// TIA Portal V16 export
// export: Created 2024-05-11T02:56:22.8632211Z, ExportSetting WithDefaults, DisplayName Totally Integrated Automation Portal, DisplayVersion V16, DisplayName TIA Portal Version Control Interface, DisplayVersion V16, DisplayName TIA Portal Openness, DisplayVersion V16, DisplayName STEP 7 Professional, DisplayVersion V16, DisplayName STEP 7 Safety, DisplayVersion V16, DisplayName WinCC Professional, DisplayVersion V16
FUNCTION_BLOCK "K06_动作"   // FB6, LAD
{ S7_Optimized_Access := 'TRUE' }
VERSION : 0.1
// stored: AutoNumber false, IsIECCheckEnabled false, IsRetainMemResEnabled false, MemoryReserve 100, SetENOAutomatically false, UDAEnableTagReadback false
   VAR
      INV_Time1 : IEC_TIMER;
      INV_Time2 : IEC_TIMER;
      F100_Val_Instance1 { S7_SetPoint := 'True'} : "F100_Val";   // EN阻挡
      F100_Val_Instance2 { S7_SetPoint := 'True'} : "F100_Val";   // EN提升机
      F100_Val_Instance3 { S7_SetPoint := 'True'} : "F100_Val";   // EX阻挡
      F100_Val_Instance4 { S7_SetPoint := 'True'} : "F100_Val";   // EX提升机
      F100_Val_Instance5 { S7_SetPoint := 'True'} : "F100_Val";   // ST01上阻挡
      F100_Val_Instance6 { S7_SetPoint := 'True'} : "F100_Val";   // ST01下阻挡
      F100_Val_Instance7 { S7_SetPoint := 'True'} : "F100_Val";   // ST02上阻挡
      F100_Val_Instance8 { S7_SetPoint := 'True'} : "F100_Val";   // ST02下阻挡
      F100_Val_Instance9 { S7_SetPoint := 'True'} : "F100_Val";   // ST03上阻挡
      F100_Val_Instance10 { S7_SetPoint := 'True'} : "F100_Val";   // ST03下阻挡
      F100_Val_Instance11 { S7_SetPoint := 'True'} : "F100_Val";   // ST04上阻挡
      F100_Val_Instance12 { S7_SetPoint := 'True'} : "F100_Val";   // ST05上阻挡
      F100_Val_Instance13 { S7_SetPoint := 'True'} : "F100_Val";   // ST06上阻挡
      F100_Val_Instance14 { S7_SetPoint := 'True'} : "F100_Val";   // ST07上阻挡
      F100_Val_Instance15 { S7_SetPoint := 'True'} : "F100_Val";   // ST08上阻挡
      F100_Val_Instance16 { S7_SetPoint := 'True'} : "F100_Val";   // ST09上阻挡
      F100_Val_Instance17 { S7_SetPoint := 'True'} : "F100_Val";   // ST10上阻挡
      F100_Val_Instance18 { S7_SetPoint := 'True'} : "F100_Val";   // ST11上阻挡
      F100_Val_Instance19 { S7_SetPoint := 'True'} : "F100_Val";   // ST12上阻挡
      F110_Inv_Instance1 { S7_SetPoint := 'True'} : "F110_Inv";   // 入口变频器
      F110_Inv_Instance2 { S7_SetPoint := 'True'} : "F110_Inv";   // 出口变频器
      F110_Inv_Instance3 { S7_SetPoint := 'True'} : "F110_Inv";   // 上层线体变频器
      F110_Inv_Instance4 { S7_SetPoint := 'True'} : "F110_Inv";   // 下层线体变频器
   END_VAR
   VAR_TEMP
      M_Pluse : Array[1..20] of Bool;
      上线体正转 : Bool;
      上线体反转 : Bool;
      上线体高速 : Bool;
      上线体低速 : Bool;
      上线体复位 : Bool;
      下线体正转 : Bool;
      下线体反转 : Bool;
      下线体高速 : Bool;
      下线体低速 : Bool;
      下线体复位 : Bool;
   END_VAR
   VAR_TEMP   // added for the SCL form of the ladder/FBD networks
      _w1 : Bool;
      _w2 : Bool;
      _w3 : Bool;
      _w4 : Bool;
      _w5 : Bool;
      _w6 : Bool;
      _w7 : Bool;
      _w8 : Bool;
      _w9 : Bool;
      _w10 : Bool;
      _w11 : Bool;
      _w12 : Bool;
   END_VAR
BEGIN

REGION Network 1: 阀1 入口阻挡
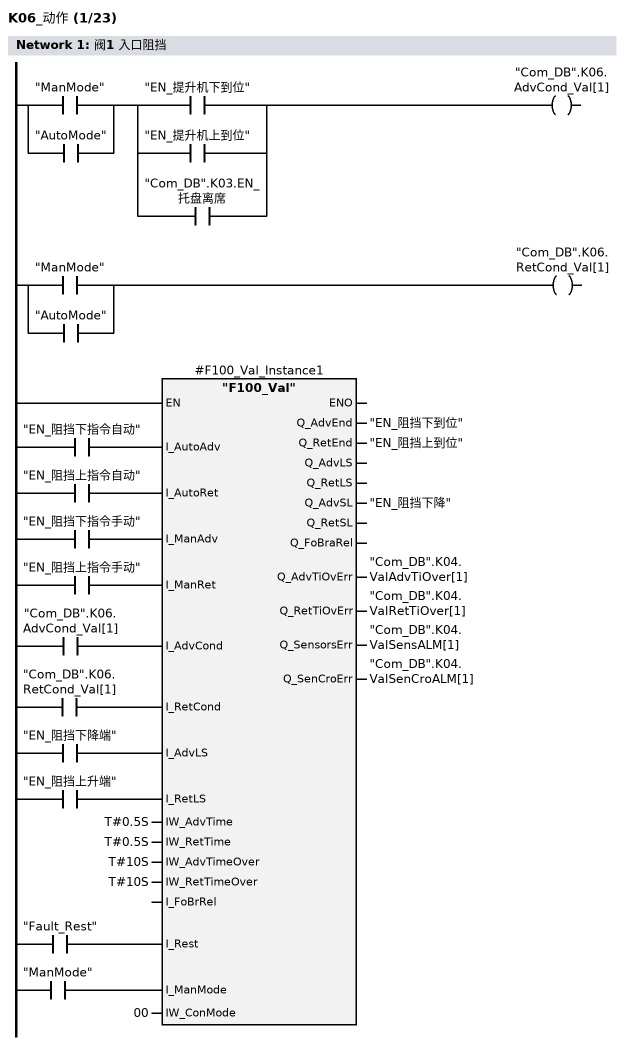
   RUNG wire#powerrail
      Contact( "ManMode" )
      wire#w1
      Contact( "EN_提升机下到位" )
      wire#w2
      Coil( "Com_DB".K06.AdvCond_Val[1] )
   END_RUNG
   RUNG wire#powerrail
      Contact( "AutoMode" )
   END_RUNG wire#w1
   RUNG wire#w1
      Contact( "EN_提升机上到位" )
   END_RUNG wire#w2
   RUNG wire#w1
      Contact( "Com_DB".K03.EN_托盘离席 )
   END_RUNG wire#w2
   RUNG wire#powerrail
      Contact( "ManMode" )
      wire#w3
      Coil( "Com_DB".K06.RetCond_Val[1] )
   END_RUNG
   RUNG wire#powerrail
      Contact( "AutoMode" )
   END_RUNG wire#w3
   RUNG wire#powerrail
      #F100_Val_Instance1(I_AutoAdv := wire#w4, I_AutoRet := wire#w5, I_ManAdv := wire#w6, I_ManRet := wire#w7, I_AdvCond := wire#w8, I_RetCond := wire#w9, I_AdvLS := wire#w10, I_RetLS := wire#w11, I_Rest := wire#w12, I_ManMode := wire#w13, IW_AdvTime := T#0.5S, IW_RetTime := T#0.5S, IW_AdvTimeOver := T#10S, IW_RetTimeOver := T#10S, I_FoBrRel :=, IW_ConMode := 00, Q_AdvEnd => "EN_阻挡下到位", Q_RetEnd => "EN_阻挡上到位", Q_AdvLS =>, Q_RetLS =>, Q_AdvSL => "EN_阻挡下降", Q_RetSL =>, Q_FoBraRel =>, Q_AdvTiOvErr => "Com_DB".K04.ValAdvTiOver[1], Q_RetTiOvErr => "Com_DB".K04.ValRetTiOver[1], Q_SensorsErr => "Com_DB".K04.ValSensALM[1], Q_SenCroErr => "Com_DB".K04.ValSenCroALM[1])
   END_RUNG
   RUNG wire#powerrail
      Contact( "EN_阻挡下指令自动" )
   END_RUNG wire#w4
   RUNG wire#powerrail
      Contact( "EN_阻挡上指令自动" )
   END_RUNG wire#w5
   RUNG wire#powerrail
      Contact( "EN_阻挡下指令手动" )
   END_RUNG wire#w6
   RUNG wire#powerrail
      Contact( "EN_阻挡上指令手动" )
   END_RUNG wire#w7
   RUNG wire#powerrail
      Contact( "Com_DB".K06.AdvCond_Val[1] )
   END_RUNG wire#w8
   RUNG wire#powerrail
      Contact( "Com_DB".K06.RetCond_Val[1] )
   END_RUNG wire#w9
   RUNG wire#powerrail
      Contact( "EN_阻挡下降端" )
   END_RUNG wire#w10
   RUNG wire#powerrail
      Contact( "EN_阻挡上升端" )
   END_RUNG wire#w11
   RUNG wire#powerrail
      Contact( "Fault_Rest" )
   END_RUNG wire#w12
   RUNG wire#powerrail
      Contact( "ManMode" )
   END_RUNG wire#w13
   // the same network as SCL:
   "Com_DB".K06.AdvCond_Val[1] := ("ManMode" OR "AutoMode") AND ("EN_提升机下到位" OR "EN_提升机上到位" OR "Com_DB".K03.EN_托盘离席);
   "Com_DB".K06.RetCond_Val[1] := "ManMode" OR "AutoMode";
   #F100_Val_Instance1(I_AutoAdv := "EN_阻挡下指令自动",   // "F100_Val"
                       I_AutoRet := "EN_阻挡上指令自动",
                       I_ManAdv := "EN_阻挡下指令手动",
                       I_ManRet := "EN_阻挡上指令手动",
                       I_AdvCond := "Com_DB".K06.AdvCond_Val[1],
                       I_RetCond := "Com_DB".K06.RetCond_Val[1],
                       I_AdvLS := "EN_阻挡下降端",
                       I_RetLS := "EN_阻挡上升端",
                       IW_AdvTime := T#0.5S,
                       IW_RetTime := T#0.5S,
                       IW_AdvTimeOver := T#10S,
                       IW_RetTimeOver := T#10S,
                       I_Rest := "Fault_Rest",
                       I_ManMode := "ManMode",
                       IW_ConMode := 00,
                       Q_AdvEnd => "EN_阻挡下到位",
                       Q_RetEnd => "EN_阻挡上到位",
                       Q_AdvSL => "EN_阻挡下降",
                       Q_AdvTiOvErr => "Com_DB".K04.ValAdvTiOver[1],
                       Q_RetTiOvErr => "Com_DB".K04.ValRetTiOver[1],
                       Q_SensorsErr => "Com_DB".K04.ValSensALM[1],
                       Q_SenCroErr => "Com_DB".K04.ValSenCroALM[1]);
END_REGION

REGION Network 2: 阀2 入口提升机
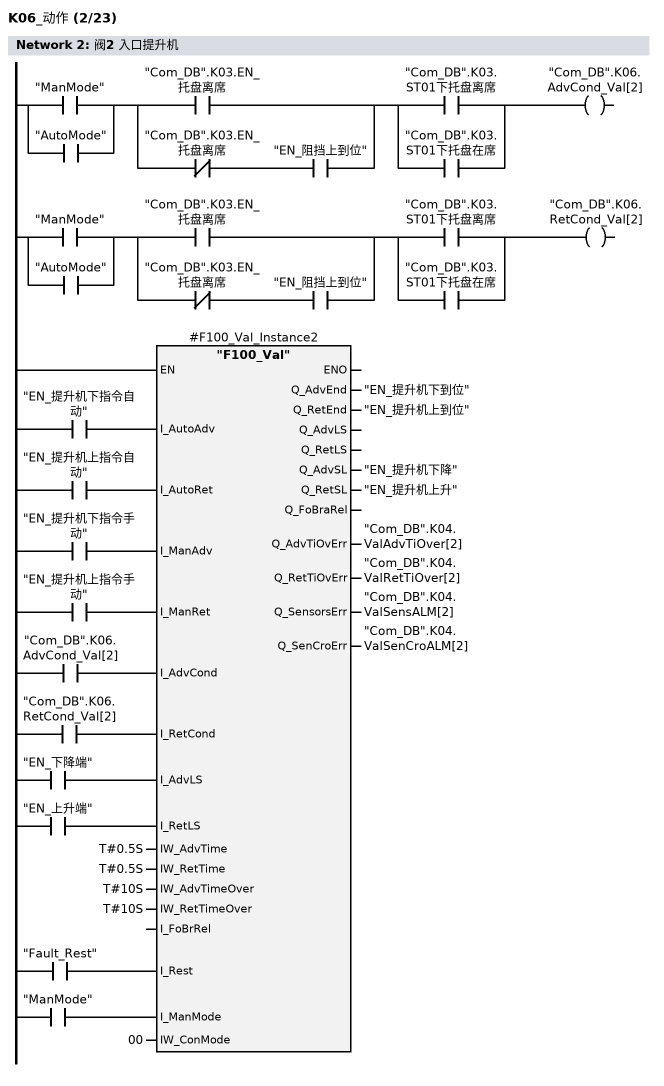
   RUNG wire#powerrail
      Contact( "ManMode" )
      wire#w1
      Contact( "Com_DB".K03.EN_托盘离席 )
      wire#w2
      Contact( "Com_DB".K03.ST01下托盘离席 )
      wire#w3
      Coil( "Com_DB".K06.AdvCond_Val[2] )
   END_RUNG
   RUNG wire#powerrail
      Contact( "AutoMode" )
   END_RUNG wire#w1
   RUNG wire#w1
      I_Contact( "Com_DB".K03.EN_托盘离席 )
      Contact( "EN_阻挡上到位" )
   END_RUNG wire#w2
   RUNG wire#w2
      Contact( "Com_DB".K03.ST01下托盘在席 )
   END_RUNG wire#w3
   RUNG wire#powerrail
      Contact( "ManMode" )
      wire#w4
      Contact( "Com_DB".K03.EN_托盘离席 )
      wire#w5
      Contact( "Com_DB".K03.ST01下托盘离席 )
      wire#w6
      Coil( "Com_DB".K06.RetCond_Val[2] )
   END_RUNG
   RUNG wire#powerrail
      Contact( "AutoMode" )
   END_RUNG wire#w4
   RUNG wire#w4
      I_Contact( "Com_DB".K03.EN_托盘离席 )
      Contact( "EN_阻挡上到位" )
   END_RUNG wire#w5
   RUNG wire#w5
      Contact( "Com_DB".K03.ST01下托盘在席 )
   END_RUNG wire#w6
   RUNG wire#powerrail
      #F100_Val_Instance2(I_AutoAdv := wire#w7, I_AutoRet := wire#w8, I_ManAdv := wire#w9, I_ManRet := wire#w10, I_AdvCond := wire#w11, I_RetCond := wire#w12, I_AdvLS := wire#w13, I_RetLS := wire#w14, I_Rest := wire#w15, I_ManMode := wire#w16, IW_AdvTime := T#0.5S, IW_RetTime := T#0.5S, IW_AdvTimeOver := T#10S, IW_RetTimeOver := T#10S, I_FoBrRel :=, IW_ConMode := 00, Q_AdvEnd => "EN_提升机下到位", Q_RetEnd => "EN_提升机上到位", Q_AdvLS =>, Q_RetLS =>, Q_AdvSL => "EN_提升机下降", Q_RetSL => "EN_提升机上升", Q_FoBraRel =>, Q_AdvTiOvErr => "Com_DB".K04.ValAdvTiOver[2], Q_RetTiOvErr => "Com_DB".K04.ValRetTiOver[2], Q_SensorsErr => "Com_DB".K04.ValSensALM[2], Q_SenCroErr => "Com_DB".K04.ValSenCroALM[2])
   END_RUNG
   RUNG wire#powerrail
      Contact( "EN_提升机下指令自动" )
   END_RUNG wire#w7
   RUNG wire#powerrail
      Contact( "EN_提升机上指令自动" )
   END_RUNG wire#w8
   RUNG wire#powerrail
      Contact( "EN_提升机下指令手动" )
   END_RUNG wire#w9
   RUNG wire#powerrail
      Contact( "EN_提升机上指令手动" )
   END_RUNG wire#w10
   RUNG wire#powerrail
      Contact( "Com_DB".K06.AdvCond_Val[2] )
   END_RUNG wire#w11
   RUNG wire#powerrail
      Contact( "Com_DB".K06.RetCond_Val[2] )
   END_RUNG wire#w12
   RUNG wire#powerrail
      Contact( "EN_下降端" )
   END_RUNG wire#w13
   RUNG wire#powerrail
      Contact( "EN_上升端" )
   END_RUNG wire#w14
   RUNG wire#powerrail
      Contact( "Fault_Rest" )
   END_RUNG wire#w15
   RUNG wire#powerrail
      Contact( "ManMode" )
   END_RUNG wire#w16
   // the same network as SCL:
   "Com_DB".K06.AdvCond_Val[2] := ("ManMode" OR "AutoMode") AND ("Com_DB".K03.EN_托盘离席 OR (NOT "Com_DB".K03.EN_托盘离席 AND "EN_阻挡上到位")) AND ("Com_DB".K03.ST01下托盘离席 OR "Com_DB".K03.ST01下托盘在席);
   "Com_DB".K06.RetCond_Val[2] := ("ManMode" OR "AutoMode") AND ("Com_DB".K03.EN_托盘离席 OR (NOT "Com_DB".K03.EN_托盘离席 AND "EN_阻挡上到位")) AND ("Com_DB".K03.ST01下托盘离席 OR "Com_DB".K03.ST01下托盘在席);
   #F100_Val_Instance2(I_AutoAdv := "EN_提升机下指令自动",   // "F100_Val"
                       I_AutoRet := "EN_提升机上指令自动",
                       I_ManAdv := "EN_提升机下指令手动",
                       I_ManRet := "EN_提升机上指令手动",
                       I_AdvCond := "Com_DB".K06.AdvCond_Val[2],
                       I_RetCond := "Com_DB".K06.RetCond_Val[2],
                       I_AdvLS := "EN_下降端",
                       I_RetLS := "EN_上升端",
                       IW_AdvTime := T#0.5S,
                       IW_RetTime := T#0.5S,
                       IW_AdvTimeOver := T#10S,
                       IW_RetTimeOver := T#10S,
                       I_Rest := "Fault_Rest",
                       I_ManMode := "ManMode",
                       IW_ConMode := 00,
                       Q_AdvEnd => "EN_提升机下到位",
                       Q_RetEnd => "EN_提升机上到位",
                       Q_AdvSL => "EN_提升机下降",
                       Q_RetSL => "EN_提升机上升",
                       Q_AdvTiOvErr => "Com_DB".K04.ValAdvTiOver[2],
                       Q_RetTiOvErr => "Com_DB".K04.ValRetTiOver[2],
                       Q_SensorsErr => "Com_DB".K04.ValSensALM[2],
                       Q_SenCroErr => "Com_DB".K04.ValSenCroALM[2]);
END_REGION

REGION Network 3: 阀3 出口阻挡
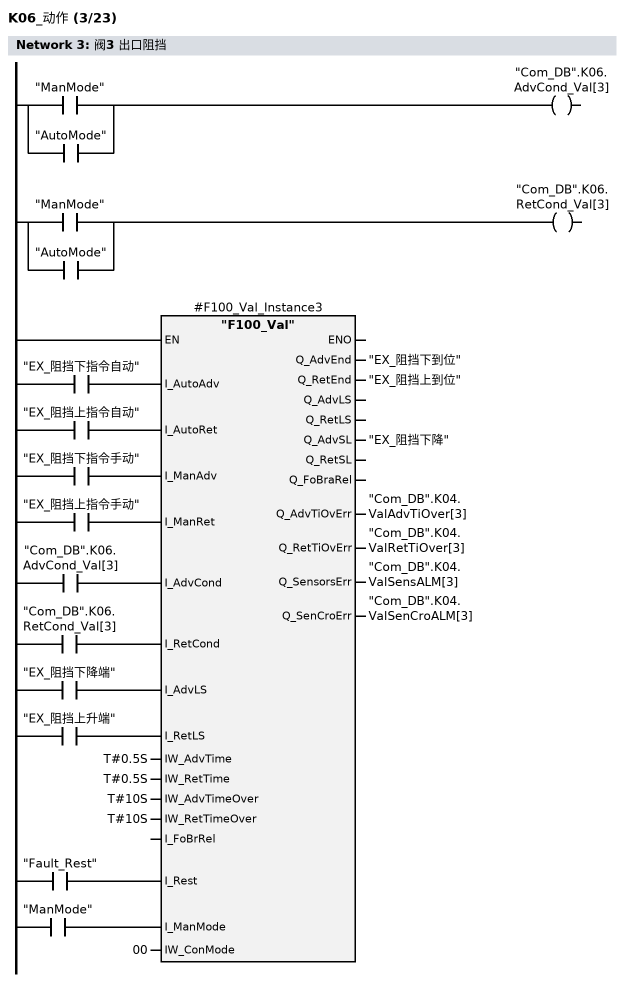
   RUNG wire#powerrail
      Contact( "ManMode" )
      wire#w1
      Coil( "Com_DB".K06.AdvCond_Val[3] )
   END_RUNG
   RUNG wire#powerrail
      Contact( "AutoMode" )
   END_RUNG wire#w1
   RUNG wire#powerrail
      Contact( "ManMode" )
      wire#w2
      Coil( "Com_DB".K06.RetCond_Val[3] )
   END_RUNG
   RUNG wire#powerrail
      Contact( "AutoMode" )
   END_RUNG wire#w2
   RUNG wire#powerrail
      #F100_Val_Instance3(I_AutoAdv := wire#w3, I_AutoRet := wire#w4, I_ManAdv := wire#w5, I_ManRet := wire#w6, I_AdvCond := wire#w7, I_RetCond := wire#w8, I_AdvLS := wire#w9, I_RetLS := wire#w10, I_Rest := wire#w11, I_ManMode := wire#w12, IW_AdvTime := T#0.5S, IW_RetTime := T#0.5S, IW_AdvTimeOver := T#10S, IW_RetTimeOver := T#10S, I_FoBrRel :=, IW_ConMode := 00, Q_AdvEnd => "EX_阻挡下到位", Q_RetEnd => "EX_阻挡上到位", Q_AdvLS =>, Q_RetLS =>, Q_AdvSL => "EX_阻挡下降", Q_RetSL =>, Q_FoBraRel =>, Q_AdvTiOvErr => "Com_DB".K04.ValAdvTiOver[3], Q_RetTiOvErr => "Com_DB".K04.ValRetTiOver[3], Q_SensorsErr => "Com_DB".K04.ValSensALM[3], Q_SenCroErr => "Com_DB".K04.ValSenCroALM[3])
   END_RUNG
   RUNG wire#powerrail
      Contact( "EX_阻挡下指令自动" )
   END_RUNG wire#w3
   RUNG wire#powerrail
      Contact( "EX_阻挡上指令自动" )
   END_RUNG wire#w4
   RUNG wire#powerrail
      Contact( "EX_阻挡下指令手动" )
   END_RUNG wire#w5
   RUNG wire#powerrail
      Contact( "EX_阻挡上指令手动" )
   END_RUNG wire#w6
   RUNG wire#powerrail
      Contact( "Com_DB".K06.AdvCond_Val[3] )
   END_RUNG wire#w7
   RUNG wire#powerrail
      Contact( "Com_DB".K06.RetCond_Val[3] )
   END_RUNG wire#w8
   RUNG wire#powerrail
      Contact( "EX_阻挡下降端" )
   END_RUNG wire#w9
   RUNG wire#powerrail
      Contact( "EX_阻挡上升端" )
   END_RUNG wire#w10
   RUNG wire#powerrail
      Contact( "Fault_Rest" )
   END_RUNG wire#w11
   RUNG wire#powerrail
      Contact( "ManMode" )
   END_RUNG wire#w12
   // the same network as SCL:
   "Com_DB".K06.AdvCond_Val[3] := "ManMode" OR "AutoMode";
   "Com_DB".K06.RetCond_Val[3] := "ManMode" OR "AutoMode";
   #F100_Val_Instance3(I_AutoAdv := "EX_阻挡下指令自动",   // "F100_Val"
                       I_AutoRet := "EX_阻挡上指令自动",
                       I_ManAdv := "EX_阻挡下指令手动",
                       I_ManRet := "EX_阻挡上指令手动",
                       I_AdvCond := "Com_DB".K06.AdvCond_Val[3],
                       I_RetCond := "Com_DB".K06.RetCond_Val[3],
                       I_AdvLS := "EX_阻挡下降端",
                       I_RetLS := "EX_阻挡上升端",
                       IW_AdvTime := T#0.5S,
                       IW_RetTime := T#0.5S,
                       IW_AdvTimeOver := T#10S,
                       IW_RetTimeOver := T#10S,
                       I_Rest := "Fault_Rest",
                       I_ManMode := "ManMode",
                       IW_ConMode := 00,
                       Q_AdvEnd => "EX_阻挡下到位",
                       Q_RetEnd => "EX_阻挡上到位",
                       Q_AdvSL => "EX_阻挡下降",
                       Q_AdvTiOvErr => "Com_DB".K04.ValAdvTiOver[3],
                       Q_RetTiOvErr => "Com_DB".K04.ValRetTiOver[3],
                       Q_SensorsErr => "Com_DB".K04.ValSensALM[3],
                       Q_SenCroErr => "Com_DB".K04.ValSenCroALM[3]);
END_REGION

REGION Network 4: 阀4 出口提升机
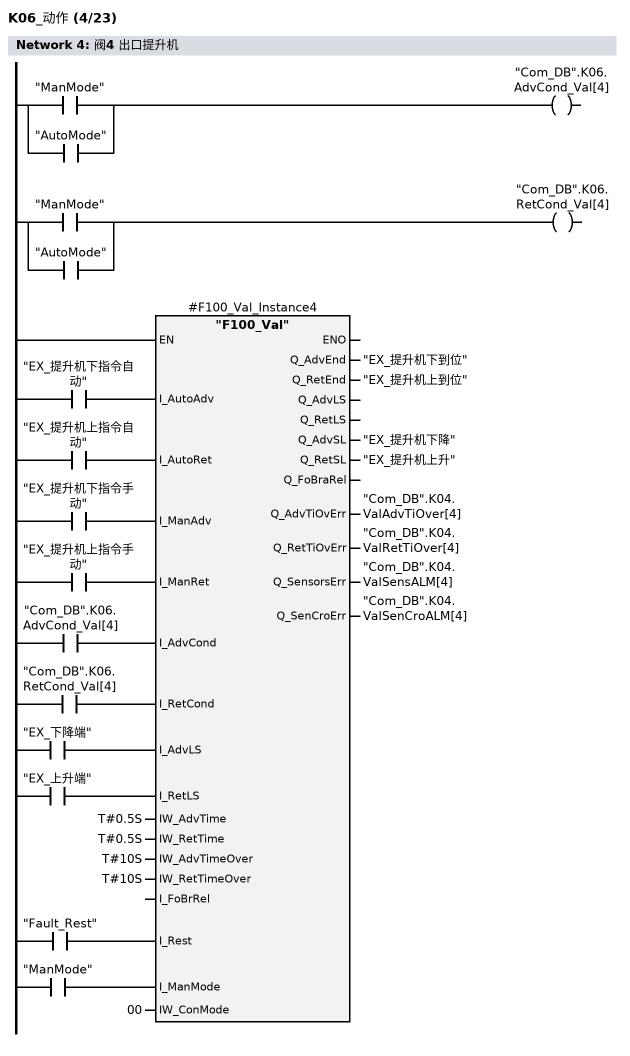
   RUNG wire#powerrail
      Contact( "ManMode" )
      wire#w1
      Coil( "Com_DB".K06.AdvCond_Val[4] )
   END_RUNG
   RUNG wire#powerrail
      Contact( "AutoMode" )
   END_RUNG wire#w1
   RUNG wire#powerrail
      Contact( "ManMode" )
      wire#w2
      Coil( "Com_DB".K06.RetCond_Val[4] )
   END_RUNG
   RUNG wire#powerrail
      Contact( "AutoMode" )
   END_RUNG wire#w2
   RUNG wire#powerrail
      #F100_Val_Instance4(I_AutoAdv := wire#w3, I_AutoRet := wire#w4, I_ManAdv := wire#w5, I_ManRet := wire#w6, I_AdvCond := wire#w7, I_RetCond := wire#w8, I_AdvLS := wire#w9, I_RetLS := wire#w10, I_Rest := wire#w11, I_ManMode := wire#w12, IW_AdvTime := T#0.5S, IW_RetTime := T#0.5S, IW_AdvTimeOver := T#10S, IW_RetTimeOver := T#10S, I_FoBrRel :=, IW_ConMode := 00, Q_AdvEnd => "EX_提升机下到位", Q_RetEnd => "EX_提升机上到位", Q_AdvLS =>, Q_RetLS =>, Q_AdvSL => "EX_提升机下降", Q_RetSL => "EX_提升机上升", Q_FoBraRel =>, Q_AdvTiOvErr => "Com_DB".K04.ValAdvTiOver[4], Q_RetTiOvErr => "Com_DB".K04.ValRetTiOver[4], Q_SensorsErr => "Com_DB".K04.ValSensALM[4], Q_SenCroErr => "Com_DB".K04.ValSenCroALM[4])
   END_RUNG
   RUNG wire#powerrail
      Contact( "EX_提升机下指令自动" )
   END_RUNG wire#w3
   RUNG wire#powerrail
      Contact( "EX_提升机上指令自动" )
   END_RUNG wire#w4
   RUNG wire#powerrail
      Contact( "EX_提升机下指令手动" )
   END_RUNG wire#w5
   RUNG wire#powerrail
      Contact( "EX_提升机上指令手动" )
   END_RUNG wire#w6
   RUNG wire#powerrail
      Contact( "Com_DB".K06.AdvCond_Val[4] )
   END_RUNG wire#w7
   RUNG wire#powerrail
      Contact( "Com_DB".K06.RetCond_Val[4] )
   END_RUNG wire#w8
   RUNG wire#powerrail
      Contact( "EX_下降端" )
   END_RUNG wire#w9
   RUNG wire#powerrail
      Contact( "EX_上升端" )
   END_RUNG wire#w10
   RUNG wire#powerrail
      Contact( "Fault_Rest" )
   END_RUNG wire#w11
   RUNG wire#powerrail
      Contact( "ManMode" )
   END_RUNG wire#w12
   // the same network as SCL:
   "Com_DB".K06.AdvCond_Val[4] := "ManMode" OR "AutoMode";
   "Com_DB".K06.RetCond_Val[4] := "ManMode" OR "AutoMode";
   #F100_Val_Instance4(I_AutoAdv := "EX_提升机下指令自动",   // "F100_Val"
                       I_AutoRet := "EX_提升机上指令自动",
                       I_ManAdv := "EX_提升机下指令手动",
                       I_ManRet := "EX_提升机上指令手动",
                       I_AdvCond := "Com_DB".K06.AdvCond_Val[4],
                       I_RetCond := "Com_DB".K06.RetCond_Val[4],
                       I_AdvLS := "EX_下降端",
                       I_RetLS := "EX_上升端",
                       IW_AdvTime := T#0.5S,
                       IW_RetTime := T#0.5S,
                       IW_AdvTimeOver := T#10S,
                       IW_RetTimeOver := T#10S,
                       I_Rest := "Fault_Rest",
                       I_ManMode := "ManMode",
                       IW_ConMode := 00,
                       Q_AdvEnd => "EX_提升机下到位",
                       Q_RetEnd => "EX_提升机上到位",
                       Q_AdvSL => "EX_提升机下降",
                       Q_RetSL => "EX_提升机上升",
                       Q_AdvTiOvErr => "Com_DB".K04.ValAdvTiOver[4],
                       Q_RetTiOvErr => "Com_DB".K04.ValRetTiOver[4],
                       Q_SensorsErr => "Com_DB".K04.ValSensALM[4],
                       Q_SenCroErr => "Com_DB".K04.ValSenCroALM[4]);
END_REGION

REGION Network 5: 阀5 ST01上阻挡
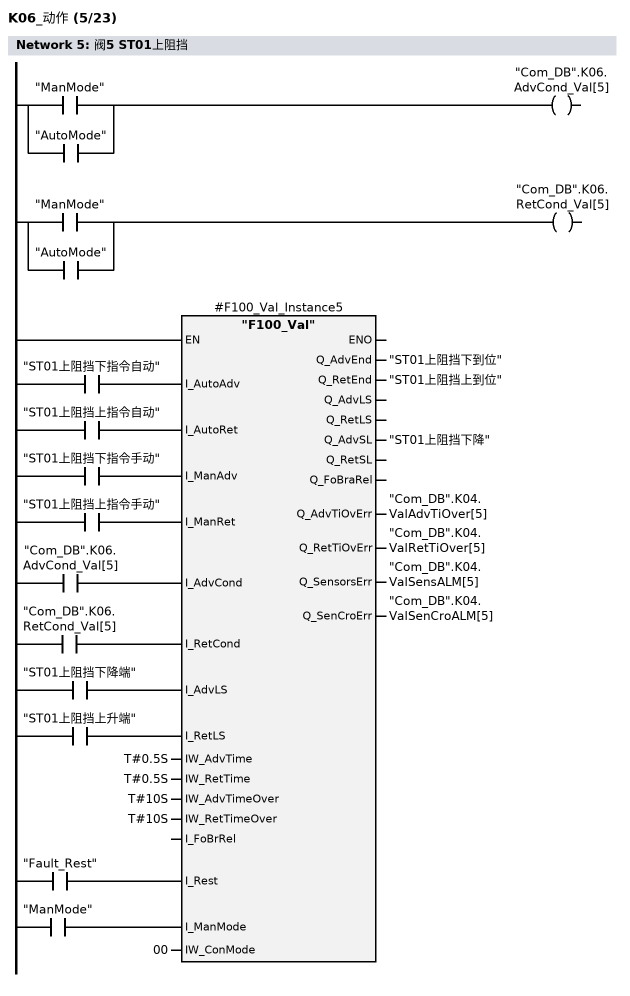
   RUNG wire#powerrail
      Contact( "ManMode" )
      wire#w1
      Coil( "Com_DB".K06.AdvCond_Val[5] )
   END_RUNG
   RUNG wire#powerrail
      Contact( "AutoMode" )
   END_RUNG wire#w1
   RUNG wire#powerrail
      Contact( "ManMode" )
      wire#w2
      Coil( "Com_DB".K06.RetCond_Val[5] )
   END_RUNG
   RUNG wire#powerrail
      Contact( "AutoMode" )
   END_RUNG wire#w2
   RUNG wire#powerrail
      #F100_Val_Instance5(I_AutoAdv := wire#w3, I_AutoRet := wire#w4, I_ManAdv := wire#w5, I_ManRet := wire#w6, I_AdvCond := wire#w7, I_RetCond := wire#w8, I_AdvLS := wire#w9, I_RetLS := wire#w10, I_Rest := wire#w11, I_ManMode := wire#w12, IW_AdvTime := T#0.5S, IW_RetTime := T#0.5S, IW_AdvTimeOver := T#10S, IW_RetTimeOver := T#10S, I_FoBrRel :=, IW_ConMode := 00, Q_AdvEnd => "ST01上阻挡下到位", Q_RetEnd => "ST01上阻挡上到位", Q_AdvLS =>, Q_RetLS =>, Q_AdvSL => "ST01上阻挡下降", Q_RetSL =>, Q_FoBraRel =>, Q_AdvTiOvErr => "Com_DB".K04.ValAdvTiOver[5], Q_RetTiOvErr => "Com_DB".K04.ValRetTiOver[5], Q_SensorsErr => "Com_DB".K04.ValSensALM[5], Q_SenCroErr => "Com_DB".K04.ValSenCroALM[5])
   END_RUNG
   RUNG wire#powerrail
      Contact( "ST01上阻挡下指令自动" )
   END_RUNG wire#w3
   RUNG wire#powerrail
      Contact( "ST01上阻挡上指令自动" )
   END_RUNG wire#w4
   RUNG wire#powerrail
      Contact( "ST01上阻挡下指令手动" )
   END_RUNG wire#w5
   RUNG wire#powerrail
      Contact( "ST01上阻挡上指令手动" )
   END_RUNG wire#w6
   RUNG wire#powerrail
      Contact( "Com_DB".K06.AdvCond_Val[5] )
   END_RUNG wire#w7
   RUNG wire#powerrail
      Contact( "Com_DB".K06.RetCond_Val[5] )
   END_RUNG wire#w8
   RUNG wire#powerrail
      Contact( "ST01上阻挡下降端" )
   END_RUNG wire#w9
   RUNG wire#powerrail
      Contact( "ST01上阻挡上升端" )
   END_RUNG wire#w10
   RUNG wire#powerrail
      Contact( "Fault_Rest" )
   END_RUNG wire#w11
   RUNG wire#powerrail
      Contact( "ManMode" )
   END_RUNG wire#w12
   // the same network as SCL:
   "Com_DB".K06.AdvCond_Val[5] := "ManMode" OR "AutoMode";
   "Com_DB".K06.RetCond_Val[5] := "ManMode" OR "AutoMode";
   #F100_Val_Instance5(I_AutoAdv := "ST01上阻挡下指令自动",   // "F100_Val"
                       I_AutoRet := "ST01上阻挡上指令自动",
                       I_ManAdv := "ST01上阻挡下指令手动",
                       I_ManRet := "ST01上阻挡上指令手动",
                       I_AdvCond := "Com_DB".K06.AdvCond_Val[5],
                       I_RetCond := "Com_DB".K06.RetCond_Val[5],
                       I_AdvLS := "ST01上阻挡下降端",
                       I_RetLS := "ST01上阻挡上升端",
                       IW_AdvTime := T#0.5S,
                       IW_RetTime := T#0.5S,
                       IW_AdvTimeOver := T#10S,
                       IW_RetTimeOver := T#10S,
                       I_Rest := "Fault_Rest",
                       I_ManMode := "ManMode",
                       IW_ConMode := 00,
                       Q_AdvEnd => "ST01上阻挡下到位",
                       Q_RetEnd => "ST01上阻挡上到位",
                       Q_AdvSL => "ST01上阻挡下降",
                       Q_AdvTiOvErr => "Com_DB".K04.ValAdvTiOver[5],
                       Q_RetTiOvErr => "Com_DB".K04.ValRetTiOver[5],
                       Q_SensorsErr => "Com_DB".K04.ValSensALM[5],
                       Q_SenCroErr => "Com_DB".K04.ValSenCroALM[5]);
END_REGION

REGION Network 6: 阀6 ST01下阻挡
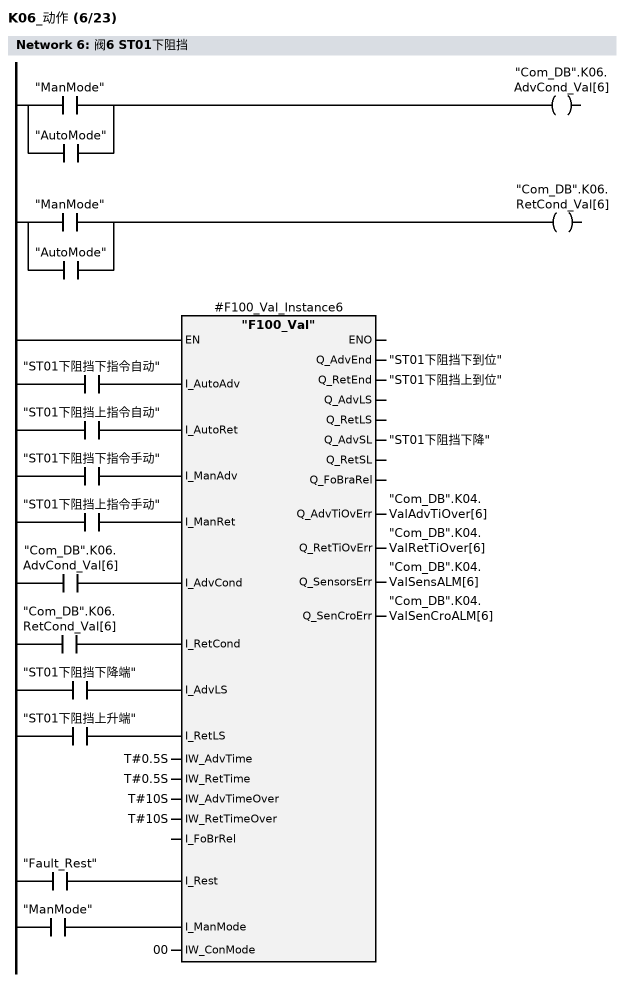
   RUNG wire#powerrail
      Contact( "ManMode" )
      wire#w1
      Coil( "Com_DB".K06.AdvCond_Val[6] )
   END_RUNG
   RUNG wire#powerrail
      Contact( "AutoMode" )
   END_RUNG wire#w1
   RUNG wire#powerrail
      Contact( "ManMode" )
      wire#w2
      Coil( "Com_DB".K06.RetCond_Val[6] )
   END_RUNG
   RUNG wire#powerrail
      Contact( "AutoMode" )
   END_RUNG wire#w2
   RUNG wire#powerrail
      #F100_Val_Instance6(I_AutoAdv := wire#w3, I_AutoRet := wire#w4, I_ManAdv := wire#w5, I_ManRet := wire#w6, I_AdvCond := wire#w7, I_RetCond := wire#w8, I_AdvLS := wire#w9, I_RetLS := wire#w10, I_Rest := wire#w11, I_ManMode := wire#w12, IW_AdvTime := T#0.5S, IW_RetTime := T#0.5S, IW_AdvTimeOver := T#10S, IW_RetTimeOver := T#10S, I_FoBrRel :=, IW_ConMode := 00, Q_AdvEnd => "ST01下阻挡下到位", Q_RetEnd => "ST01下阻挡上到位", Q_AdvLS =>, Q_RetLS =>, Q_AdvSL => "ST01下阻挡下降", Q_RetSL =>, Q_FoBraRel =>, Q_AdvTiOvErr => "Com_DB".K04.ValAdvTiOver[6], Q_RetTiOvErr => "Com_DB".K04.ValRetTiOver[6], Q_SensorsErr => "Com_DB".K04.ValSensALM[6], Q_SenCroErr => "Com_DB".K04.ValSenCroALM[6])
   END_RUNG
   RUNG wire#powerrail
      Contact( "ST01下阻挡下指令自动" )
   END_RUNG wire#w3
   RUNG wire#powerrail
      Contact( "ST01下阻挡上指令自动" )
   END_RUNG wire#w4
   RUNG wire#powerrail
      Contact( "ST01下阻挡下指令手动" )
   END_RUNG wire#w5
   RUNG wire#powerrail
      Contact( "ST01下阻挡上指令手动" )
   END_RUNG wire#w6
   RUNG wire#powerrail
      Contact( "Com_DB".K06.AdvCond_Val[6] )
   END_RUNG wire#w7
   RUNG wire#powerrail
      Contact( "Com_DB".K06.RetCond_Val[6] )
   END_RUNG wire#w8
   RUNG wire#powerrail
      Contact( "ST01下阻挡下降端" )
   END_RUNG wire#w9
   RUNG wire#powerrail
      Contact( "ST01下阻挡上升端" )
   END_RUNG wire#w10
   RUNG wire#powerrail
      Contact( "Fault_Rest" )
   END_RUNG wire#w11
   RUNG wire#powerrail
      Contact( "ManMode" )
   END_RUNG wire#w12
   // the same network as SCL:
   "Com_DB".K06.AdvCond_Val[6] := "ManMode" OR "AutoMode";
   "Com_DB".K06.RetCond_Val[6] := "ManMode" OR "AutoMode";
   #F100_Val_Instance6(I_AutoAdv := "ST01下阻挡下指令自动",   // "F100_Val"
                       I_AutoRet := "ST01下阻挡上指令自动",
                       I_ManAdv := "ST01下阻挡下指令手动",
                       I_ManRet := "ST01下阻挡上指令手动",
                       I_AdvCond := "Com_DB".K06.AdvCond_Val[6],
                       I_RetCond := "Com_DB".K06.RetCond_Val[6],
                       I_AdvLS := "ST01下阻挡下降端",
                       I_RetLS := "ST01下阻挡上升端",
                       IW_AdvTime := T#0.5S,
                       IW_RetTime := T#0.5S,
                       IW_AdvTimeOver := T#10S,
                       IW_RetTimeOver := T#10S,
                       I_Rest := "Fault_Rest",
                       I_ManMode := "ManMode",
                       IW_ConMode := 00,
                       Q_AdvEnd => "ST01下阻挡下到位",
                       Q_RetEnd => "ST01下阻挡上到位",
                       Q_AdvSL => "ST01下阻挡下降",
                       Q_AdvTiOvErr => "Com_DB".K04.ValAdvTiOver[6],
                       Q_RetTiOvErr => "Com_DB".K04.ValRetTiOver[6],
                       Q_SensorsErr => "Com_DB".K04.ValSensALM[6],
                       Q_SenCroErr => "Com_DB".K04.ValSenCroALM[6]);
END_REGION

REGION Network 7: 阀7 ST02上阻挡
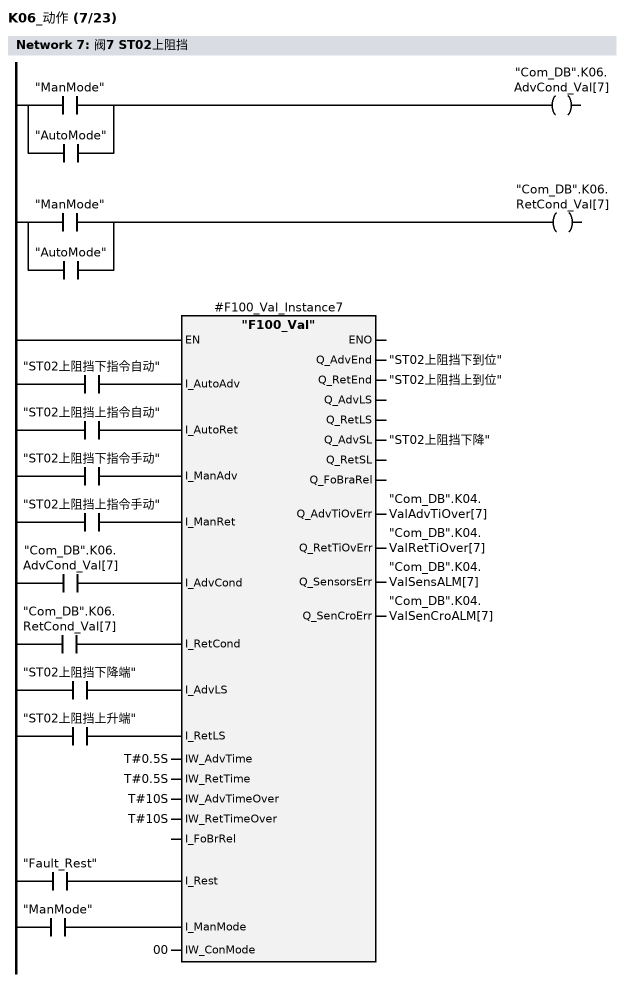
   RUNG wire#powerrail
      Contact( "ManMode" )
      wire#w1
      Coil( "Com_DB".K06.AdvCond_Val[7] )
   END_RUNG
   RUNG wire#powerrail
      Contact( "AutoMode" )
   END_RUNG wire#w1
   RUNG wire#powerrail
      Contact( "ManMode" )
      wire#w2
      Coil( "Com_DB".K06.RetCond_Val[7] )
   END_RUNG
   RUNG wire#powerrail
      Contact( "AutoMode" )
   END_RUNG wire#w2
   RUNG wire#powerrail
      #F100_Val_Instance7(I_AutoAdv := wire#w3, I_AutoRet := wire#w4, I_ManAdv := wire#w5, I_ManRet := wire#w6, I_AdvCond := wire#w7, I_RetCond := wire#w8, I_AdvLS := wire#w9, I_RetLS := wire#w10, I_Rest := wire#w11, I_ManMode := wire#w12, IW_AdvTime := T#0.5S, IW_RetTime := T#0.5S, IW_AdvTimeOver := T#10S, IW_RetTimeOver := T#10S, I_FoBrRel :=, IW_ConMode := 00, Q_AdvEnd => "ST02上阻挡下到位", Q_RetEnd => "ST02上阻挡上到位", Q_AdvLS =>, Q_RetLS =>, Q_AdvSL => "ST02上阻挡下降", Q_RetSL =>, Q_FoBraRel =>, Q_AdvTiOvErr => "Com_DB".K04.ValAdvTiOver[7], Q_RetTiOvErr => "Com_DB".K04.ValRetTiOver[7], Q_SensorsErr => "Com_DB".K04.ValSensALM[7], Q_SenCroErr => "Com_DB".K04.ValSenCroALM[7])
   END_RUNG
   RUNG wire#powerrail
      Contact( "ST02上阻挡下指令自动" )
   END_RUNG wire#w3
   RUNG wire#powerrail
      Contact( "ST02上阻挡上指令自动" )
   END_RUNG wire#w4
   RUNG wire#powerrail
      Contact( "ST02上阻挡下指令手动" )
   END_RUNG wire#w5
   RUNG wire#powerrail
      Contact( "ST02上阻挡上指令手动" )
   END_RUNG wire#w6
   RUNG wire#powerrail
      Contact( "Com_DB".K06.AdvCond_Val[7] )
   END_RUNG wire#w7
   RUNG wire#powerrail
      Contact( "Com_DB".K06.RetCond_Val[7] )
   END_RUNG wire#w8
   RUNG wire#powerrail
      Contact( "ST02上阻挡下降端" )
   END_RUNG wire#w9
   RUNG wire#powerrail
      Contact( "ST02上阻挡上升端" )
   END_RUNG wire#w10
   RUNG wire#powerrail
      Contact( "Fault_Rest" )
   END_RUNG wire#w11
   RUNG wire#powerrail
      Contact( "ManMode" )
   END_RUNG wire#w12
   // the same network as SCL:
   "Com_DB".K06.AdvCond_Val[7] := "ManMode" OR "AutoMode";
   "Com_DB".K06.RetCond_Val[7] := "ManMode" OR "AutoMode";
   #F100_Val_Instance7(I_AutoAdv := "ST02上阻挡下指令自动",   // "F100_Val"
                       I_AutoRet := "ST02上阻挡上指令自动",
                       I_ManAdv := "ST02上阻挡下指令手动",
                       I_ManRet := "ST02上阻挡上指令手动",
                       I_AdvCond := "Com_DB".K06.AdvCond_Val[7],
                       I_RetCond := "Com_DB".K06.RetCond_Val[7],
                       I_AdvLS := "ST02上阻挡下降端",
                       I_RetLS := "ST02上阻挡上升端",
                       IW_AdvTime := T#0.5S,
                       IW_RetTime := T#0.5S,
                       IW_AdvTimeOver := T#10S,
                       IW_RetTimeOver := T#10S,
                       I_Rest := "Fault_Rest",
                       I_ManMode := "ManMode",
                       IW_ConMode := 00,
                       Q_AdvEnd => "ST02上阻挡下到位",
                       Q_RetEnd => "ST02上阻挡上到位",
                       Q_AdvSL => "ST02上阻挡下降",
                       Q_AdvTiOvErr => "Com_DB".K04.ValAdvTiOver[7],
                       Q_RetTiOvErr => "Com_DB".K04.ValRetTiOver[7],
                       Q_SensorsErr => "Com_DB".K04.ValSensALM[7],
                       Q_SenCroErr => "Com_DB".K04.ValSenCroALM[7]);
END_REGION

REGION Network 8: 阀8 ST02下阻挡
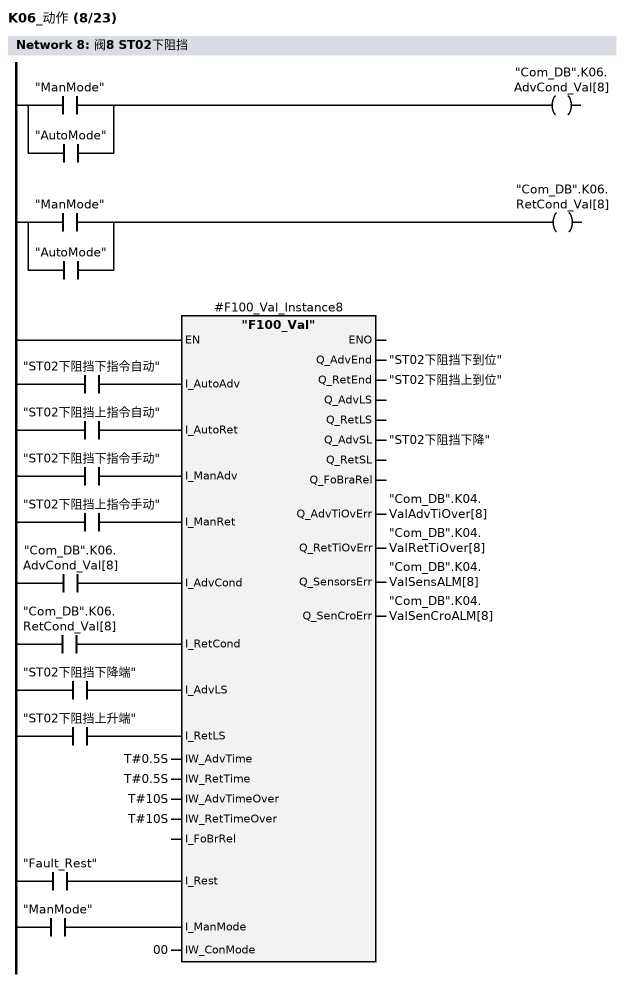
   RUNG wire#powerrail
      Contact( "ManMode" )
      wire#w1
      Coil( "Com_DB".K06.AdvCond_Val[8] )
   END_RUNG
   RUNG wire#powerrail
      Contact( "AutoMode" )
   END_RUNG wire#w1
   RUNG wire#powerrail
      Contact( "ManMode" )
      wire#w2
      Coil( "Com_DB".K06.RetCond_Val[8] )
   END_RUNG
   RUNG wire#powerrail
      Contact( "AutoMode" )
   END_RUNG wire#w2
   RUNG wire#powerrail
      #F100_Val_Instance8(I_AutoAdv := wire#w3, I_AutoRet := wire#w4, I_ManAdv := wire#w5, I_ManRet := wire#w6, I_AdvCond := wire#w7, I_RetCond := wire#w8, I_AdvLS := wire#w9, I_RetLS := wire#w10, I_Rest := wire#w11, I_ManMode := wire#w12, IW_AdvTime := T#0.5S, IW_RetTime := T#0.5S, IW_AdvTimeOver := T#10S, IW_RetTimeOver := T#10S, I_FoBrRel :=, IW_ConMode := 00, Q_AdvEnd => "ST02下阻挡下到位", Q_RetEnd => "ST02下阻挡上到位", Q_AdvLS =>, Q_RetLS =>, Q_AdvSL => "ST02下阻挡下降", Q_RetSL =>, Q_FoBraRel =>, Q_AdvTiOvErr => "Com_DB".K04.ValAdvTiOver[8], Q_RetTiOvErr => "Com_DB".K04.ValRetTiOver[8], Q_SensorsErr => "Com_DB".K04.ValSensALM[8], Q_SenCroErr => "Com_DB".K04.ValSenCroALM[8])
   END_RUNG
   RUNG wire#powerrail
      Contact( "ST02下阻挡下指令自动" )
   END_RUNG wire#w3
   RUNG wire#powerrail
      Contact( "ST02下阻挡上指令自动" )
   END_RUNG wire#w4
   RUNG wire#powerrail
      Contact( "ST02下阻挡下指令手动" )
   END_RUNG wire#w5
   RUNG wire#powerrail
      Contact( "ST02下阻挡上指令手动" )
   END_RUNG wire#w6
   RUNG wire#powerrail
      Contact( "Com_DB".K06.AdvCond_Val[8] )
   END_RUNG wire#w7
   RUNG wire#powerrail
      Contact( "Com_DB".K06.RetCond_Val[8] )
   END_RUNG wire#w8
   RUNG wire#powerrail
      Contact( "ST02下阻挡下降端" )
   END_RUNG wire#w9
   RUNG wire#powerrail
      Contact( "ST02下阻挡上升端" )
   END_RUNG wire#w10
   RUNG wire#powerrail
      Contact( "Fault_Rest" )
   END_RUNG wire#w11
   RUNG wire#powerrail
      Contact( "ManMode" )
   END_RUNG wire#w12
   // the same network as SCL:
   "Com_DB".K06.AdvCond_Val[8] := "ManMode" OR "AutoMode";
   "Com_DB".K06.RetCond_Val[8] := "ManMode" OR "AutoMode";
   #F100_Val_Instance8(I_AutoAdv := "ST02下阻挡下指令自动",   // "F100_Val"
                       I_AutoRet := "ST02下阻挡上指令自动",
                       I_ManAdv := "ST02下阻挡下指令手动",
                       I_ManRet := "ST02下阻挡上指令手动",
                       I_AdvCond := "Com_DB".K06.AdvCond_Val[8],
                       I_RetCond := "Com_DB".K06.RetCond_Val[8],
                       I_AdvLS := "ST02下阻挡下降端",
                       I_RetLS := "ST02下阻挡上升端",
                       IW_AdvTime := T#0.5S,
                       IW_RetTime := T#0.5S,
                       IW_AdvTimeOver := T#10S,
                       IW_RetTimeOver := T#10S,
                       I_Rest := "Fault_Rest",
                       I_ManMode := "ManMode",
                       IW_ConMode := 00,
                       Q_AdvEnd => "ST02下阻挡下到位",
                       Q_RetEnd => "ST02下阻挡上到位",
                       Q_AdvSL => "ST02下阻挡下降",
                       Q_AdvTiOvErr => "Com_DB".K04.ValAdvTiOver[8],
                       Q_RetTiOvErr => "Com_DB".K04.ValRetTiOver[8],
                       Q_SensorsErr => "Com_DB".K04.ValSensALM[8],
                       Q_SenCroErr => "Com_DB".K04.ValSenCroALM[8]);
END_REGION

REGION Network 9: 阀9 ST03上阻挡
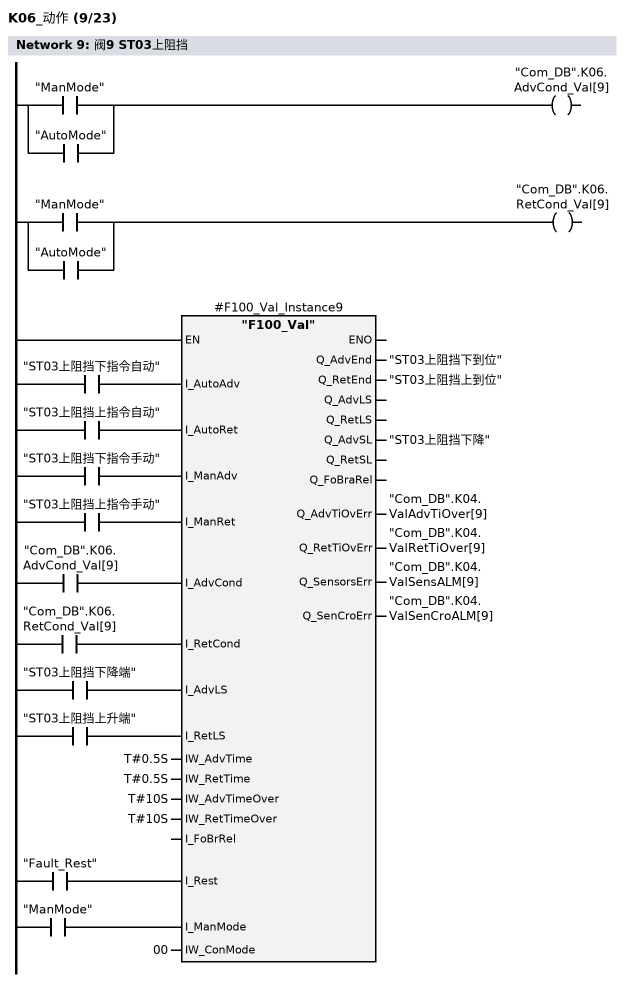
   RUNG wire#powerrail
      Contact( "ManMode" )
      wire#w1
      Coil( "Com_DB".K06.AdvCond_Val[9] )
   END_RUNG
   RUNG wire#powerrail
      Contact( "AutoMode" )
   END_RUNG wire#w1
   RUNG wire#powerrail
      Contact( "ManMode" )
      wire#w2
      Coil( "Com_DB".K06.RetCond_Val[9] )
   END_RUNG
   RUNG wire#powerrail
      Contact( "AutoMode" )
   END_RUNG wire#w2
   RUNG wire#powerrail
      #F100_Val_Instance9(I_AutoAdv := wire#w3, I_AutoRet := wire#w4, I_ManAdv := wire#w5, I_ManRet := wire#w6, I_AdvCond := wire#w7, I_RetCond := wire#w8, I_AdvLS := wire#w9, I_RetLS := wire#w10, I_Rest := wire#w11, I_ManMode := wire#w12, IW_AdvTime := T#0.5S, IW_RetTime := T#0.5S, IW_AdvTimeOver := T#10S, IW_RetTimeOver := T#10S, I_FoBrRel :=, IW_ConMode := 00, Q_AdvEnd => "ST03上阻挡下到位", Q_RetEnd => "ST03上阻挡上到位", Q_AdvLS =>, Q_RetLS =>, Q_AdvSL => "ST03上阻挡下降", Q_RetSL =>, Q_FoBraRel =>, Q_AdvTiOvErr => "Com_DB".K04.ValAdvTiOver[9], Q_RetTiOvErr => "Com_DB".K04.ValRetTiOver[9], Q_SensorsErr => "Com_DB".K04.ValSensALM[9], Q_SenCroErr => "Com_DB".K04.ValSenCroALM[9])
   END_RUNG
   RUNG wire#powerrail
      Contact( "ST03上阻挡下指令自动" )
   END_RUNG wire#w3
   RUNG wire#powerrail
      Contact( "ST03上阻挡上指令自动" )
   END_RUNG wire#w4
   RUNG wire#powerrail
      Contact( "ST03上阻挡下指令手动" )
   END_RUNG wire#w5
   RUNG wire#powerrail
      Contact( "ST03上阻挡上指令手动" )
   END_RUNG wire#w6
   RUNG wire#powerrail
      Contact( "Com_DB".K06.AdvCond_Val[9] )
   END_RUNG wire#w7
   RUNG wire#powerrail
      Contact( "Com_DB".K06.RetCond_Val[9] )
   END_RUNG wire#w8
   RUNG wire#powerrail
      Contact( "ST03上阻挡下降端" )
   END_RUNG wire#w9
   RUNG wire#powerrail
      Contact( "ST03上阻挡上升端" )
   END_RUNG wire#w10
   RUNG wire#powerrail
      Contact( "Fault_Rest" )
   END_RUNG wire#w11
   RUNG wire#powerrail
      Contact( "ManMode" )
   END_RUNG wire#w12
   // the same network as SCL:
   "Com_DB".K06.AdvCond_Val[9] := "ManMode" OR "AutoMode";
   "Com_DB".K06.RetCond_Val[9] := "ManMode" OR "AutoMode";
   #F100_Val_Instance9(I_AutoAdv := "ST03上阻挡下指令自动",   // "F100_Val"
                       I_AutoRet := "ST03上阻挡上指令自动",
                       I_ManAdv := "ST03上阻挡下指令手动",
                       I_ManRet := "ST03上阻挡上指令手动",
                       I_AdvCond := "Com_DB".K06.AdvCond_Val[9],
                       I_RetCond := "Com_DB".K06.RetCond_Val[9],
                       I_AdvLS := "ST03上阻挡下降端",
                       I_RetLS := "ST03上阻挡上升端",
                       IW_AdvTime := T#0.5S,
                       IW_RetTime := T#0.5S,
                       IW_AdvTimeOver := T#10S,
                       IW_RetTimeOver := T#10S,
                       I_Rest := "Fault_Rest",
                       I_ManMode := "ManMode",
                       IW_ConMode := 00,
                       Q_AdvEnd => "ST03上阻挡下到位",
                       Q_RetEnd => "ST03上阻挡上到位",
                       Q_AdvSL => "ST03上阻挡下降",
                       Q_AdvTiOvErr => "Com_DB".K04.ValAdvTiOver[9],
                       Q_RetTiOvErr => "Com_DB".K04.ValRetTiOver[9],
                       Q_SensorsErr => "Com_DB".K04.ValSensALM[9],
                       Q_SenCroErr => "Com_DB".K04.ValSenCroALM[9]);
END_REGION

REGION Network 10: 阀10 ST03下阻挡
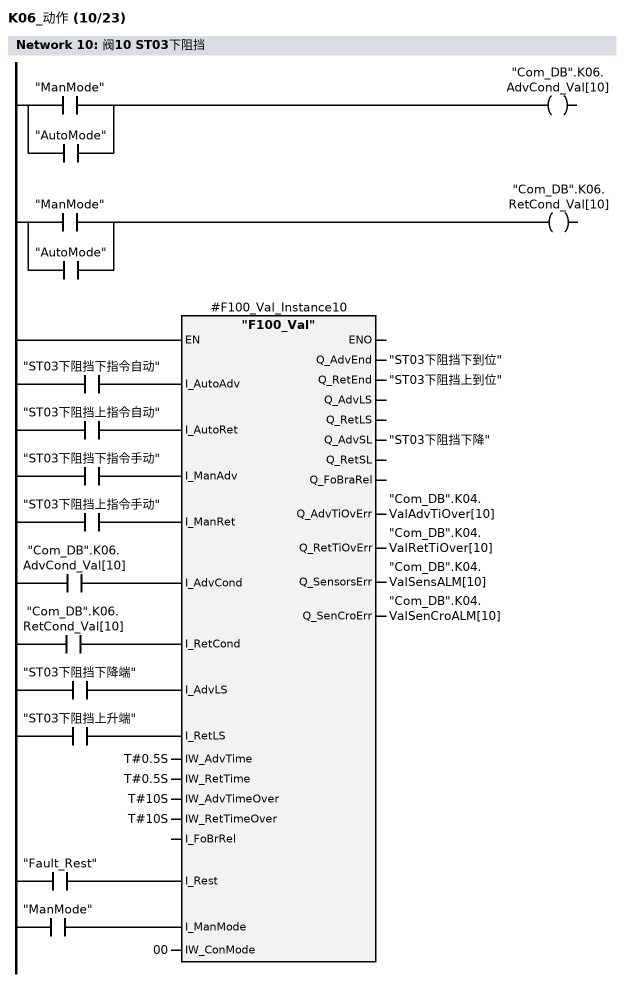
   RUNG wire#powerrail
      Contact( "ManMode" )
      wire#w1
      Coil( "Com_DB".K06.AdvCond_Val[10] )
   END_RUNG
   RUNG wire#powerrail
      Contact( "AutoMode" )
   END_RUNG wire#w1
   RUNG wire#powerrail
      Contact( "ManMode" )
      wire#w2
      Coil( "Com_DB".K06.RetCond_Val[10] )
   END_RUNG
   RUNG wire#powerrail
      Contact( "AutoMode" )
   END_RUNG wire#w2
   RUNG wire#powerrail
      #F100_Val_Instance10(I_AutoAdv := wire#w3, I_AutoRet := wire#w4, I_ManAdv := wire#w5, I_ManRet := wire#w6, I_AdvCond := wire#w7, I_RetCond := wire#w8, I_AdvLS := wire#w9, I_RetLS := wire#w10, I_Rest := wire#w11, I_ManMode := wire#w12, IW_AdvTime := T#0.5S, IW_RetTime := T#0.5S, IW_AdvTimeOver := T#10S, IW_RetTimeOver := T#10S, I_FoBrRel :=, IW_ConMode := 00, Q_AdvEnd => "ST03下阻挡下到位", Q_RetEnd => "ST03下阻挡上到位", Q_AdvLS =>, Q_RetLS =>, Q_AdvSL => "ST03下阻挡下降", Q_RetSL =>, Q_FoBraRel =>, Q_AdvTiOvErr => "Com_DB".K04.ValAdvTiOver[10], Q_RetTiOvErr => "Com_DB".K04.ValRetTiOver[10], Q_SensorsErr => "Com_DB".K04.ValSensALM[10], Q_SenCroErr => "Com_DB".K04.ValSenCroALM[10])
   END_RUNG
   RUNG wire#powerrail
      Contact( "ST03下阻挡下指令自动" )
   END_RUNG wire#w3
   RUNG wire#powerrail
      Contact( "ST03下阻挡上指令自动" )
   END_RUNG wire#w4
   RUNG wire#powerrail
      Contact( "ST03下阻挡下指令手动" )
   END_RUNG wire#w5
   RUNG wire#powerrail
      Contact( "ST03下阻挡上指令手动" )
   END_RUNG wire#w6
   RUNG wire#powerrail
      Contact( "Com_DB".K06.AdvCond_Val[10] )
   END_RUNG wire#w7
   RUNG wire#powerrail
      Contact( "Com_DB".K06.RetCond_Val[10] )
   END_RUNG wire#w8
   RUNG wire#powerrail
      Contact( "ST03下阻挡下降端" )
   END_RUNG wire#w9
   RUNG wire#powerrail
      Contact( "ST03下阻挡上升端" )
   END_RUNG wire#w10
   RUNG wire#powerrail
      Contact( "Fault_Rest" )
   END_RUNG wire#w11
   RUNG wire#powerrail
      Contact( "ManMode" )
   END_RUNG wire#w12
   // the same network as SCL:
   "Com_DB".K06.AdvCond_Val[10] := "ManMode" OR "AutoMode";
   "Com_DB".K06.RetCond_Val[10] := "ManMode" OR "AutoMode";
   #F100_Val_Instance10(I_AutoAdv := "ST03下阻挡下指令自动",   // "F100_Val"
                        I_AutoRet := "ST03下阻挡上指令自动",
                        I_ManAdv := "ST03下阻挡下指令手动",
                        I_ManRet := "ST03下阻挡上指令手动",
                        I_AdvCond := "Com_DB".K06.AdvCond_Val[10],
                        I_RetCond := "Com_DB".K06.RetCond_Val[10],
                        I_AdvLS := "ST03下阻挡下降端",
                        I_RetLS := "ST03下阻挡上升端",
                        IW_AdvTime := T#0.5S,
                        IW_RetTime := T#0.5S,
                        IW_AdvTimeOver := T#10S,
                        IW_RetTimeOver := T#10S,
                        I_Rest := "Fault_Rest",
                        I_ManMode := "ManMode",
                        IW_ConMode := 00,
                        Q_AdvEnd => "ST03下阻挡下到位",
                        Q_RetEnd => "ST03下阻挡上到位",
                        Q_AdvSL => "ST03下阻挡下降",
                        Q_AdvTiOvErr => "Com_DB".K04.ValAdvTiOver[10],
                        Q_RetTiOvErr => "Com_DB".K04.ValRetTiOver[10],
                        Q_SensorsErr => "Com_DB".K04.ValSensALM[10],
                        Q_SenCroErr => "Com_DB".K04.ValSenCroALM[10]);
END_REGION

REGION Network 11: 阀11 ST04上阻挡
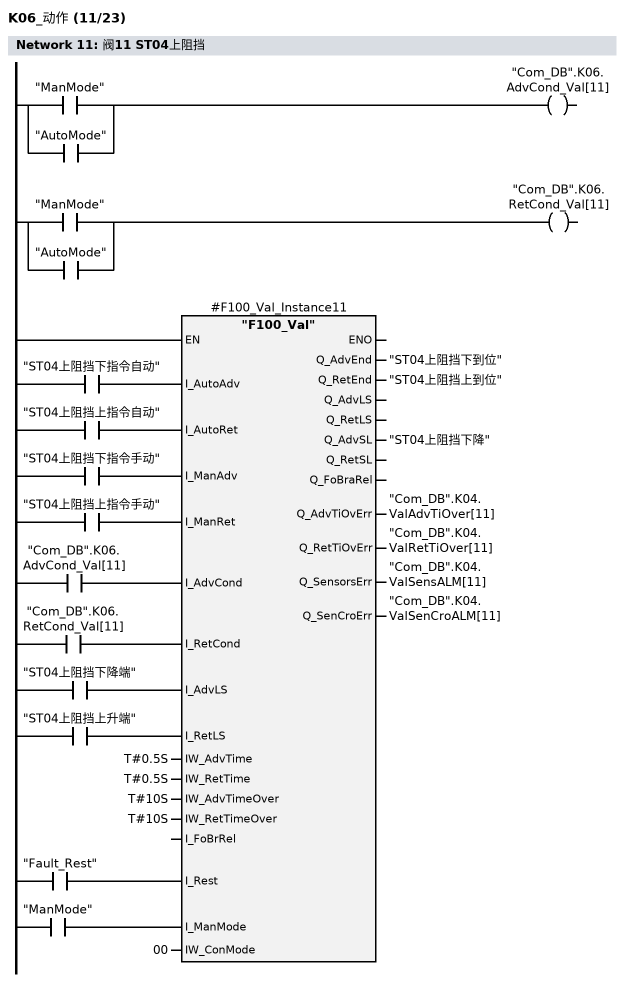
   RUNG wire#powerrail
      Contact( "ManMode" )
      wire#w1
      Coil( "Com_DB".K06.AdvCond_Val[11] )
   END_RUNG
   RUNG wire#powerrail
      Contact( "AutoMode" )
   END_RUNG wire#w1
   RUNG wire#powerrail
      Contact( "ManMode" )
      wire#w2
      Coil( "Com_DB".K06.RetCond_Val[11] )
   END_RUNG
   RUNG wire#powerrail
      Contact( "AutoMode" )
   END_RUNG wire#w2
   RUNG wire#powerrail
      #F100_Val_Instance11(I_AutoAdv := wire#w3, I_AutoRet := wire#w4, I_ManAdv := wire#w5, I_ManRet := wire#w6, I_AdvCond := wire#w7, I_RetCond := wire#w8, I_AdvLS := wire#w9, I_RetLS := wire#w10, I_Rest := wire#w11, I_ManMode := wire#w12, IW_AdvTime := T#0.5S, IW_RetTime := T#0.5S, IW_AdvTimeOver := T#10S, IW_RetTimeOver := T#10S, I_FoBrRel :=, IW_ConMode := 00, Q_AdvEnd => "ST04上阻挡下到位", Q_RetEnd => "ST04上阻挡上到位", Q_AdvLS =>, Q_RetLS =>, Q_AdvSL => "ST04上阻挡下降", Q_RetSL =>, Q_FoBraRel =>, Q_AdvTiOvErr => "Com_DB".K04.ValAdvTiOver[11], Q_RetTiOvErr => "Com_DB".K04.ValRetTiOver[11], Q_SensorsErr => "Com_DB".K04.ValSensALM[11], Q_SenCroErr => "Com_DB".K04.ValSenCroALM[11])
   END_RUNG
   RUNG wire#powerrail
      Contact( "ST04上阻挡下指令自动" )
   END_RUNG wire#w3
   RUNG wire#powerrail
      Contact( "ST04上阻挡上指令自动" )
   END_RUNG wire#w4
   RUNG wire#powerrail
      Contact( "ST04上阻挡下指令手动" )
   END_RUNG wire#w5
   RUNG wire#powerrail
      Contact( "ST04上阻挡上指令手动" )
   END_RUNG wire#w6
   RUNG wire#powerrail
      Contact( "Com_DB".K06.AdvCond_Val[11] )
   END_RUNG wire#w7
   RUNG wire#powerrail
      Contact( "Com_DB".K06.RetCond_Val[11] )
   END_RUNG wire#w8
   RUNG wire#powerrail
      Contact( "ST04上阻挡下降端" )
   END_RUNG wire#w9
   RUNG wire#powerrail
      Contact( "ST04上阻挡上升端" )
   END_RUNG wire#w10
   RUNG wire#powerrail
      Contact( "Fault_Rest" )
   END_RUNG wire#w11
   RUNG wire#powerrail
      Contact( "ManMode" )
   END_RUNG wire#w12
   // the same network as SCL:
   "Com_DB".K06.AdvCond_Val[11] := "ManMode" OR "AutoMode";
   "Com_DB".K06.RetCond_Val[11] := "ManMode" OR "AutoMode";
   #F100_Val_Instance11(I_AutoAdv := "ST04上阻挡下指令自动",   // "F100_Val"
                        I_AutoRet := "ST04上阻挡上指令自动",
                        I_ManAdv := "ST04上阻挡下指令手动",
                        I_ManRet := "ST04上阻挡上指令手动",
                        I_AdvCond := "Com_DB".K06.AdvCond_Val[11],
                        I_RetCond := "Com_DB".K06.RetCond_Val[11],
                        I_AdvLS := "ST04上阻挡下降端",
                        I_RetLS := "ST04上阻挡上升端",
                        IW_AdvTime := T#0.5S,
                        IW_RetTime := T#0.5S,
                        IW_AdvTimeOver := T#10S,
                        IW_RetTimeOver := T#10S,
                        I_Rest := "Fault_Rest",
                        I_ManMode := "ManMode",
                        IW_ConMode := 00,
                        Q_AdvEnd => "ST04上阻挡下到位",
                        Q_RetEnd => "ST04上阻挡上到位",
                        Q_AdvSL => "ST04上阻挡下降",
                        Q_AdvTiOvErr => "Com_DB".K04.ValAdvTiOver[11],
                        Q_RetTiOvErr => "Com_DB".K04.ValRetTiOver[11],
                        Q_SensorsErr => "Com_DB".K04.ValSensALM[11],
                        Q_SenCroErr => "Com_DB".K04.ValSenCroALM[11]);
END_REGION

REGION Network 12: 阀12 ST05上阻挡
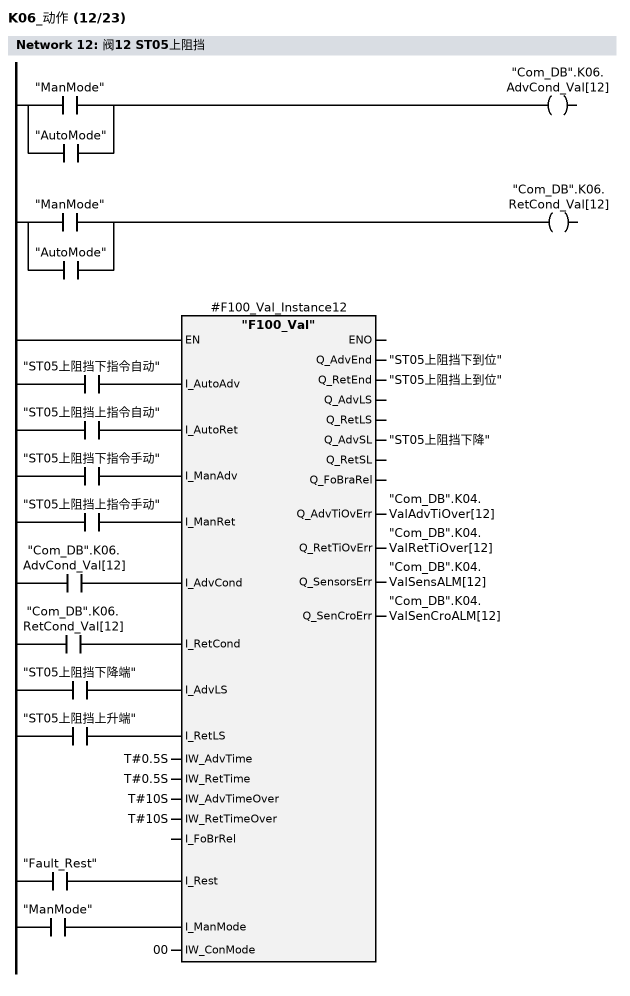
   RUNG wire#powerrail
      Contact( "ManMode" )
      wire#w1
      Coil( "Com_DB".K06.AdvCond_Val[12] )
   END_RUNG
   RUNG wire#powerrail
      Contact( "AutoMode" )
   END_RUNG wire#w1
   RUNG wire#powerrail
      Contact( "ManMode" )
      wire#w2
      Coil( "Com_DB".K06.RetCond_Val[12] )
   END_RUNG
   RUNG wire#powerrail
      Contact( "AutoMode" )
   END_RUNG wire#w2
   RUNG wire#powerrail
      #F100_Val_Instance12(I_AutoAdv := wire#w3, I_AutoRet := wire#w4, I_ManAdv := wire#w5, I_ManRet := wire#w6, I_AdvCond := wire#w7, I_RetCond := wire#w8, I_AdvLS := wire#w9, I_RetLS := wire#w10, I_Rest := wire#w11, I_ManMode := wire#w12, IW_AdvTime := T#0.5S, IW_RetTime := T#0.5S, IW_AdvTimeOver := T#10S, IW_RetTimeOver := T#10S, I_FoBrRel :=, IW_ConMode := 00, Q_AdvEnd => "ST05上阻挡下到位", Q_RetEnd => "ST05上阻挡上到位", Q_AdvLS =>, Q_RetLS =>, Q_AdvSL => "ST05上阻挡下降", Q_RetSL =>, Q_FoBraRel =>, Q_AdvTiOvErr => "Com_DB".K04.ValAdvTiOver[12], Q_RetTiOvErr => "Com_DB".K04.ValRetTiOver[12], Q_SensorsErr => "Com_DB".K04.ValSensALM[12], Q_SenCroErr => "Com_DB".K04.ValSenCroALM[12])
   END_RUNG
   RUNG wire#powerrail
      Contact( "ST05上阻挡下指令自动" )
   END_RUNG wire#w3
   RUNG wire#powerrail
      Contact( "ST05上阻挡上指令自动" )
   END_RUNG wire#w4
   RUNG wire#powerrail
      Contact( "ST05上阻挡下指令手动" )
   END_RUNG wire#w5
   RUNG wire#powerrail
      Contact( "ST05上阻挡上指令手动" )
   END_RUNG wire#w6
   RUNG wire#powerrail
      Contact( "Com_DB".K06.AdvCond_Val[12] )
   END_RUNG wire#w7
   RUNG wire#powerrail
      Contact( "Com_DB".K06.RetCond_Val[12] )
   END_RUNG wire#w8
   RUNG wire#powerrail
      Contact( "ST05上阻挡下降端" )
   END_RUNG wire#w9
   RUNG wire#powerrail
      Contact( "ST05上阻挡上升端" )
   END_RUNG wire#w10
   RUNG wire#powerrail
      Contact( "Fault_Rest" )
   END_RUNG wire#w11
   RUNG wire#powerrail
      Contact( "ManMode" )
   END_RUNG wire#w12
   // the same network as SCL:
   "Com_DB".K06.AdvCond_Val[12] := "ManMode" OR "AutoMode";
   "Com_DB".K06.RetCond_Val[12] := "ManMode" OR "AutoMode";
   #F100_Val_Instance12(I_AutoAdv := "ST05上阻挡下指令自动",   // "F100_Val"
                        I_AutoRet := "ST05上阻挡上指令自动",
                        I_ManAdv := "ST05上阻挡下指令手动",
                        I_ManRet := "ST05上阻挡上指令手动",
                        I_AdvCond := "Com_DB".K06.AdvCond_Val[12],
                        I_RetCond := "Com_DB".K06.RetCond_Val[12],
                        I_AdvLS := "ST05上阻挡下降端",
                        I_RetLS := "ST05上阻挡上升端",
                        IW_AdvTime := T#0.5S,
                        IW_RetTime := T#0.5S,
                        IW_AdvTimeOver := T#10S,
                        IW_RetTimeOver := T#10S,
                        I_Rest := "Fault_Rest",
                        I_ManMode := "ManMode",
                        IW_ConMode := 00,
                        Q_AdvEnd => "ST05上阻挡下到位",
                        Q_RetEnd => "ST05上阻挡上到位",
                        Q_AdvSL => "ST05上阻挡下降",
                        Q_AdvTiOvErr => "Com_DB".K04.ValAdvTiOver[12],
                        Q_RetTiOvErr => "Com_DB".K04.ValRetTiOver[12],
                        Q_SensorsErr => "Com_DB".K04.ValSensALM[12],
                        Q_SenCroErr => "Com_DB".K04.ValSenCroALM[12]);
END_REGION

REGION Network 13: 阀13 ST06上阻挡
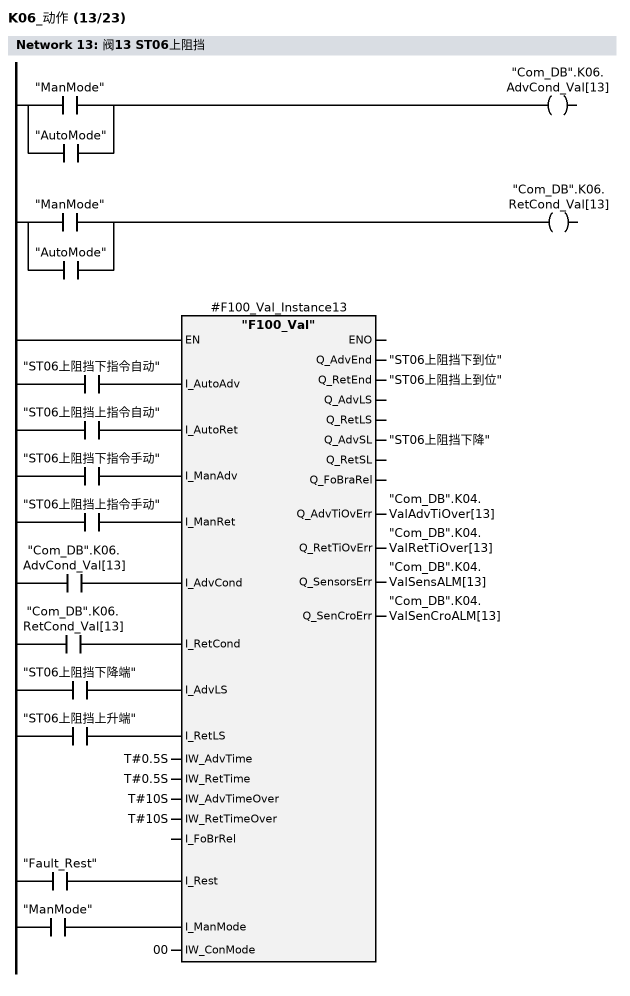
   RUNG wire#powerrail
      Contact( "ManMode" )
      wire#w1
      Coil( "Com_DB".K06.AdvCond_Val[13] )
   END_RUNG
   RUNG wire#powerrail
      Contact( "AutoMode" )
   END_RUNG wire#w1
   RUNG wire#powerrail
      Contact( "ManMode" )
      wire#w2
      Coil( "Com_DB".K06.RetCond_Val[13] )
   END_RUNG
   RUNG wire#powerrail
      Contact( "AutoMode" )
   END_RUNG wire#w2
   RUNG wire#powerrail
      #F100_Val_Instance13(I_AutoAdv := wire#w3, I_AutoRet := wire#w4, I_ManAdv := wire#w5, I_ManRet := wire#w6, I_AdvCond := wire#w7, I_RetCond := wire#w8, I_AdvLS := wire#w9, I_RetLS := wire#w10, I_Rest := wire#w11, I_ManMode := wire#w12, IW_AdvTime := T#0.5S, IW_RetTime := T#0.5S, IW_AdvTimeOver := T#10S, IW_RetTimeOver := T#10S, I_FoBrRel :=, IW_ConMode := 00, Q_AdvEnd => "ST06上阻挡下到位", Q_RetEnd => "ST06上阻挡上到位", Q_AdvLS =>, Q_RetLS =>, Q_AdvSL => "ST06上阻挡下降", Q_RetSL =>, Q_FoBraRel =>, Q_AdvTiOvErr => "Com_DB".K04.ValAdvTiOver[13], Q_RetTiOvErr => "Com_DB".K04.ValRetTiOver[13], Q_SensorsErr => "Com_DB".K04.ValSensALM[13], Q_SenCroErr => "Com_DB".K04.ValSenCroALM[13])
   END_RUNG
   RUNG wire#powerrail
      Contact( "ST06上阻挡下指令自动" )
   END_RUNG wire#w3
   RUNG wire#powerrail
      Contact( "ST06上阻挡上指令自动" )
   END_RUNG wire#w4
   RUNG wire#powerrail
      Contact( "ST06上阻挡下指令手动" )
   END_RUNG wire#w5
   RUNG wire#powerrail
      Contact( "ST06上阻挡上指令手动" )
   END_RUNG wire#w6
   RUNG wire#powerrail
      Contact( "Com_DB".K06.AdvCond_Val[13] )
   END_RUNG wire#w7
   RUNG wire#powerrail
      Contact( "Com_DB".K06.RetCond_Val[13] )
   END_RUNG wire#w8
   RUNG wire#powerrail
      Contact( "ST06上阻挡下降端" )
   END_RUNG wire#w9
   RUNG wire#powerrail
      Contact( "ST06上阻挡上升端" )
   END_RUNG wire#w10
   RUNG wire#powerrail
      Contact( "Fault_Rest" )
   END_RUNG wire#w11
   RUNG wire#powerrail
      Contact( "ManMode" )
   END_RUNG wire#w12
   // the same network as SCL:
   "Com_DB".K06.AdvCond_Val[13] := "ManMode" OR "AutoMode";
   "Com_DB".K06.RetCond_Val[13] := "ManMode" OR "AutoMode";
   #F100_Val_Instance13(I_AutoAdv := "ST06上阻挡下指令自动",   // "F100_Val"
                        I_AutoRet := "ST06上阻挡上指令自动",
                        I_ManAdv := "ST06上阻挡下指令手动",
                        I_ManRet := "ST06上阻挡上指令手动",
                        I_AdvCond := "Com_DB".K06.AdvCond_Val[13],
                        I_RetCond := "Com_DB".K06.RetCond_Val[13],
                        I_AdvLS := "ST06上阻挡下降端",
                        I_RetLS := "ST06上阻挡上升端",
                        IW_AdvTime := T#0.5S,
                        IW_RetTime := T#0.5S,
                        IW_AdvTimeOver := T#10S,
                        IW_RetTimeOver := T#10S,
                        I_Rest := "Fault_Rest",
                        I_ManMode := "ManMode",
                        IW_ConMode := 00,
                        Q_AdvEnd => "ST06上阻挡下到位",
                        Q_RetEnd => "ST06上阻挡上到位",
                        Q_AdvSL => "ST06上阻挡下降",
                        Q_AdvTiOvErr => "Com_DB".K04.ValAdvTiOver[13],
                        Q_RetTiOvErr => "Com_DB".K04.ValRetTiOver[13],
                        Q_SensorsErr => "Com_DB".K04.ValSensALM[13],
                        Q_SenCroErr => "Com_DB".K04.ValSenCroALM[13]);
END_REGION

REGION Network 14: 阀14 ST07上阻挡
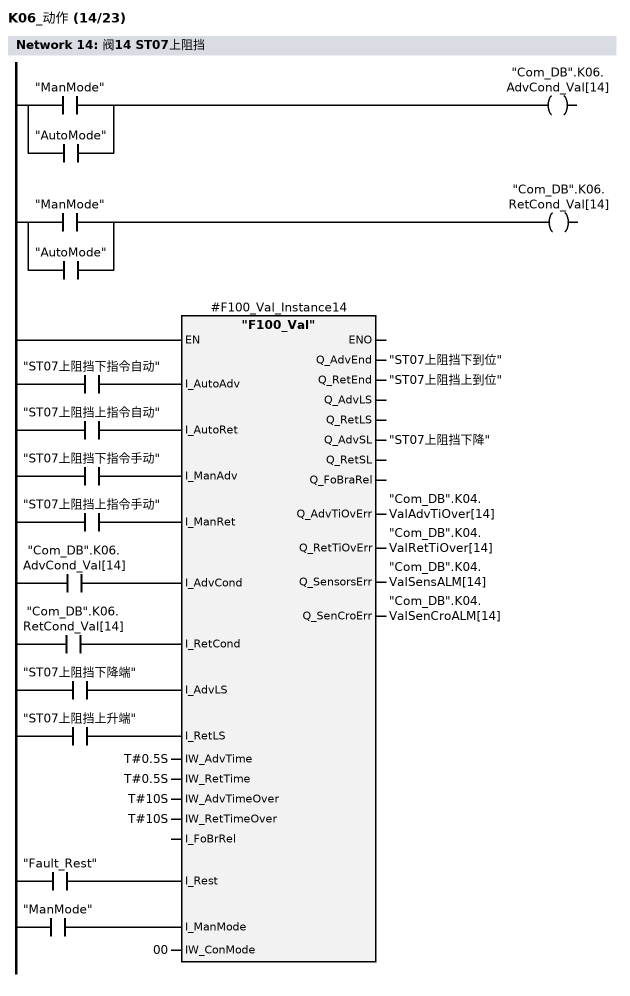
   RUNG wire#powerrail
      Contact( "ManMode" )
      wire#w1
      Coil( "Com_DB".K06.AdvCond_Val[14] )
   END_RUNG
   RUNG wire#powerrail
      Contact( "AutoMode" )
   END_RUNG wire#w1
   RUNG wire#powerrail
      Contact( "ManMode" )
      wire#w2
      Coil( "Com_DB".K06.RetCond_Val[14] )
   END_RUNG
   RUNG wire#powerrail
      Contact( "AutoMode" )
   END_RUNG wire#w2
   RUNG wire#powerrail
      #F100_Val_Instance14(I_AutoAdv := wire#w3, I_AutoRet := wire#w4, I_ManAdv := wire#w5, I_ManRet := wire#w6, I_AdvCond := wire#w7, I_RetCond := wire#w8, I_AdvLS := wire#w9, I_RetLS := wire#w10, I_Rest := wire#w11, I_ManMode := wire#w12, IW_AdvTime := T#0.5S, IW_RetTime := T#0.5S, IW_AdvTimeOver := T#10S, IW_RetTimeOver := T#10S, I_FoBrRel :=, IW_ConMode := 00, Q_AdvEnd => "ST07上阻挡下到位", Q_RetEnd => "ST07上阻挡上到位", Q_AdvLS =>, Q_RetLS =>, Q_AdvSL => "ST07上阻挡下降", Q_RetSL =>, Q_FoBraRel =>, Q_AdvTiOvErr => "Com_DB".K04.ValAdvTiOver[14], Q_RetTiOvErr => "Com_DB".K04.ValRetTiOver[14], Q_SensorsErr => "Com_DB".K04.ValSensALM[14], Q_SenCroErr => "Com_DB".K04.ValSenCroALM[14])
   END_RUNG
   RUNG wire#powerrail
      Contact( "ST07上阻挡下指令自动" )
   END_RUNG wire#w3
   RUNG wire#powerrail
      Contact( "ST07上阻挡上指令自动" )
   END_RUNG wire#w4
   RUNG wire#powerrail
      Contact( "ST07上阻挡下指令手动" )
   END_RUNG wire#w5
   RUNG wire#powerrail
      Contact( "ST07上阻挡上指令手动" )
   END_RUNG wire#w6
   RUNG wire#powerrail
      Contact( "Com_DB".K06.AdvCond_Val[14] )
   END_RUNG wire#w7
   RUNG wire#powerrail
      Contact( "Com_DB".K06.RetCond_Val[14] )
   END_RUNG wire#w8
   RUNG wire#powerrail
      Contact( "ST07上阻挡下降端" )
   END_RUNG wire#w9
   RUNG wire#powerrail
      Contact( "ST07上阻挡上升端" )
   END_RUNG wire#w10
   RUNG wire#powerrail
      Contact( "Fault_Rest" )
   END_RUNG wire#w11
   RUNG wire#powerrail
      Contact( "ManMode" )
   END_RUNG wire#w12
   // the same network as SCL:
   "Com_DB".K06.AdvCond_Val[14] := "ManMode" OR "AutoMode";
   "Com_DB".K06.RetCond_Val[14] := "ManMode" OR "AutoMode";
   #F100_Val_Instance14(I_AutoAdv := "ST07上阻挡下指令自动",   // "F100_Val"
                        I_AutoRet := "ST07上阻挡上指令自动",
                        I_ManAdv := "ST07上阻挡下指令手动",
                        I_ManRet := "ST07上阻挡上指令手动",
                        I_AdvCond := "Com_DB".K06.AdvCond_Val[14],
                        I_RetCond := "Com_DB".K06.RetCond_Val[14],
                        I_AdvLS := "ST07上阻挡下降端",
                        I_RetLS := "ST07上阻挡上升端",
                        IW_AdvTime := T#0.5S,
                        IW_RetTime := T#0.5S,
                        IW_AdvTimeOver := T#10S,
                        IW_RetTimeOver := T#10S,
                        I_Rest := "Fault_Rest",
                        I_ManMode := "ManMode",
                        IW_ConMode := 00,
                        Q_AdvEnd => "ST07上阻挡下到位",
                        Q_RetEnd => "ST07上阻挡上到位",
                        Q_AdvSL => "ST07上阻挡下降",
                        Q_AdvTiOvErr => "Com_DB".K04.ValAdvTiOver[14],
                        Q_RetTiOvErr => "Com_DB".K04.ValRetTiOver[14],
                        Q_SensorsErr => "Com_DB".K04.ValSensALM[14],
                        Q_SenCroErr => "Com_DB".K04.ValSenCroALM[14]);
END_REGION

REGION Network 15: 阀15 ST08上阻挡
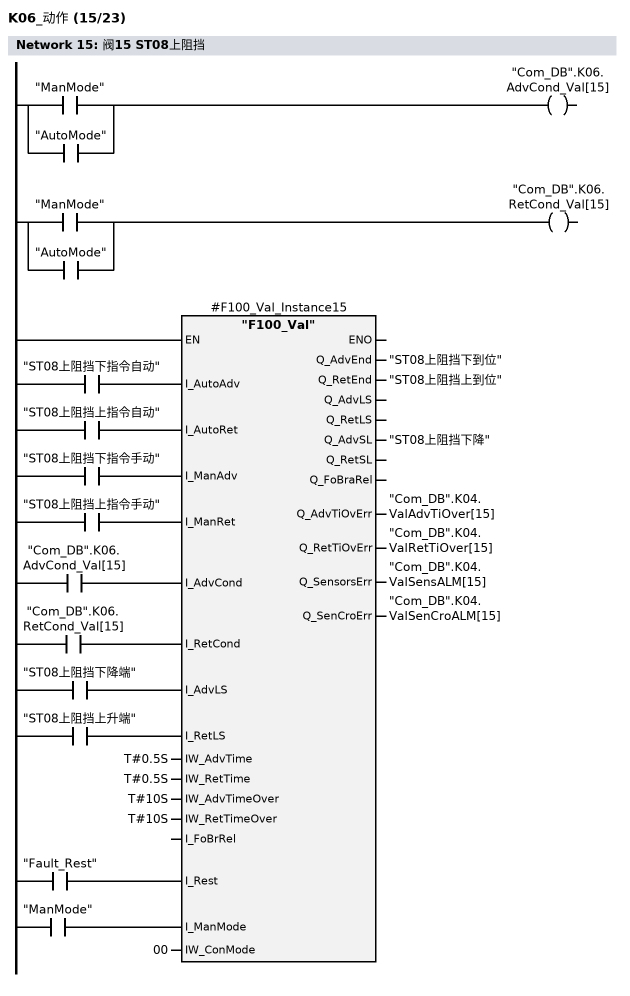
   RUNG wire#powerrail
      Contact( "ManMode" )
      wire#w1
      Coil( "Com_DB".K06.AdvCond_Val[15] )
   END_RUNG
   RUNG wire#powerrail
      Contact( "AutoMode" )
   END_RUNG wire#w1
   RUNG wire#powerrail
      Contact( "ManMode" )
      wire#w2
      Coil( "Com_DB".K06.RetCond_Val[15] )
   END_RUNG
   RUNG wire#powerrail
      Contact( "AutoMode" )
   END_RUNG wire#w2
   RUNG wire#powerrail
      #F100_Val_Instance15(I_AutoAdv := wire#w3, I_AutoRet := wire#w4, I_ManAdv := wire#w5, I_ManRet := wire#w6, I_AdvCond := wire#w7, I_RetCond := wire#w8, I_AdvLS := wire#w9, I_RetLS := wire#w10, I_Rest := wire#w11, I_ManMode := wire#w12, IW_AdvTime := T#0.5S, IW_RetTime := T#0.5S, IW_AdvTimeOver := T#10S, IW_RetTimeOver := T#10S, I_FoBrRel :=, IW_ConMode := 00, Q_AdvEnd => "ST08上阻挡下到位", Q_RetEnd => "ST08上阻挡上到位", Q_AdvLS =>, Q_RetLS =>, Q_AdvSL => "ST08上阻挡下降", Q_RetSL =>, Q_FoBraRel =>, Q_AdvTiOvErr => "Com_DB".K04.ValAdvTiOver[15], Q_RetTiOvErr => "Com_DB".K04.ValRetTiOver[15], Q_SensorsErr => "Com_DB".K04.ValSensALM[15], Q_SenCroErr => "Com_DB".K04.ValSenCroALM[15])
   END_RUNG
   RUNG wire#powerrail
      Contact( "ST08上阻挡下指令自动" )
   END_RUNG wire#w3
   RUNG wire#powerrail
      Contact( "ST08上阻挡上指令自动" )
   END_RUNG wire#w4
   RUNG wire#powerrail
      Contact( "ST08上阻挡下指令手动" )
   END_RUNG wire#w5
   RUNG wire#powerrail
      Contact( "ST08上阻挡上指令手动" )
   END_RUNG wire#w6
   RUNG wire#powerrail
      Contact( "Com_DB".K06.AdvCond_Val[15] )
   END_RUNG wire#w7
   RUNG wire#powerrail
      Contact( "Com_DB".K06.RetCond_Val[15] )
   END_RUNG wire#w8
   RUNG wire#powerrail
      Contact( "ST08上阻挡下降端" )
   END_RUNG wire#w9
   RUNG wire#powerrail
      Contact( "ST08上阻挡上升端" )
   END_RUNG wire#w10
   RUNG wire#powerrail
      Contact( "Fault_Rest" )
   END_RUNG wire#w11
   RUNG wire#powerrail
      Contact( "ManMode" )
   END_RUNG wire#w12
   // the same network as SCL:
   "Com_DB".K06.AdvCond_Val[15] := "ManMode" OR "AutoMode";
   "Com_DB".K06.RetCond_Val[15] := "ManMode" OR "AutoMode";
   #F100_Val_Instance15(I_AutoAdv := "ST08上阻挡下指令自动",   // "F100_Val"
                        I_AutoRet := "ST08上阻挡上指令自动",
                        I_ManAdv := "ST08上阻挡下指令手动",
                        I_ManRet := "ST08上阻挡上指令手动",
                        I_AdvCond := "Com_DB".K06.AdvCond_Val[15],
                        I_RetCond := "Com_DB".K06.RetCond_Val[15],
                        I_AdvLS := "ST08上阻挡下降端",
                        I_RetLS := "ST08上阻挡上升端",
                        IW_AdvTime := T#0.5S,
                        IW_RetTime := T#0.5S,
                        IW_AdvTimeOver := T#10S,
                        IW_RetTimeOver := T#10S,
                        I_Rest := "Fault_Rest",
                        I_ManMode := "ManMode",
                        IW_ConMode := 00,
                        Q_AdvEnd => "ST08上阻挡下到位",
                        Q_RetEnd => "ST08上阻挡上到位",
                        Q_AdvSL => "ST08上阻挡下降",
                        Q_AdvTiOvErr => "Com_DB".K04.ValAdvTiOver[15],
                        Q_RetTiOvErr => "Com_DB".K04.ValRetTiOver[15],
                        Q_SensorsErr => "Com_DB".K04.ValSensALM[15],
                        Q_SenCroErr => "Com_DB".K04.ValSenCroALM[15]);
END_REGION

REGION Network 16: 阀16 ST09上阻挡
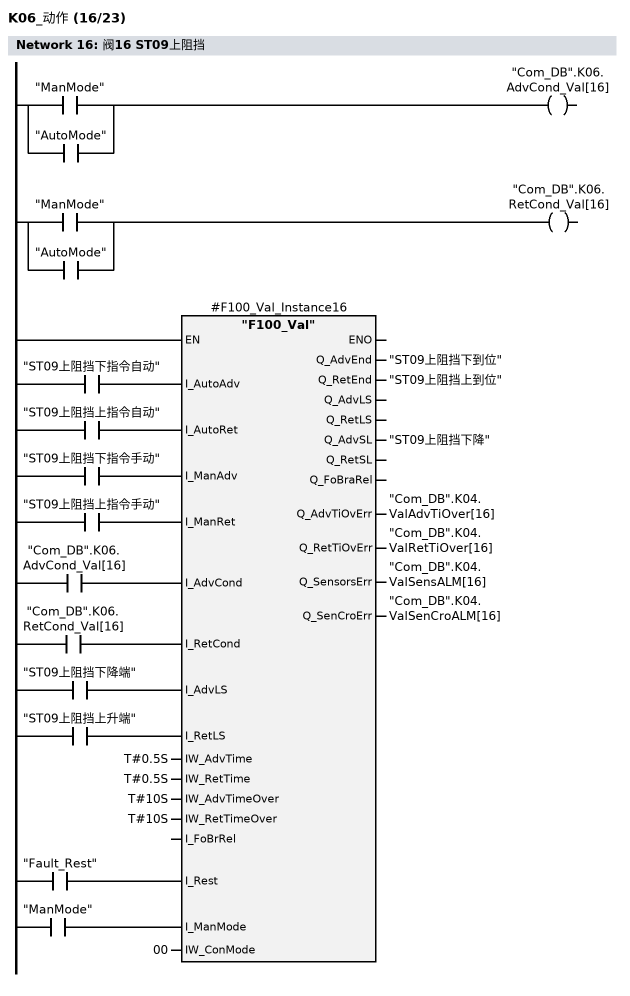
   RUNG wire#powerrail
      Contact( "ManMode" )
      wire#w1
      Coil( "Com_DB".K06.AdvCond_Val[16] )
   END_RUNG
   RUNG wire#powerrail
      Contact( "AutoMode" )
   END_RUNG wire#w1
   RUNG wire#powerrail
      Contact( "ManMode" )
      wire#w2
      Coil( "Com_DB".K06.RetCond_Val[16] )
   END_RUNG
   RUNG wire#powerrail
      Contact( "AutoMode" )
   END_RUNG wire#w2
   RUNG wire#powerrail
      #F100_Val_Instance16(I_AutoAdv := wire#w3, I_AutoRet := wire#w4, I_ManAdv := wire#w5, I_ManRet := wire#w6, I_AdvCond := wire#w7, I_RetCond := wire#w8, I_AdvLS := wire#w9, I_RetLS := wire#w10, I_Rest := wire#w11, I_ManMode := wire#w12, IW_AdvTime := T#0.5S, IW_RetTime := T#0.5S, IW_AdvTimeOver := T#10S, IW_RetTimeOver := T#10S, I_FoBrRel :=, IW_ConMode := 00, Q_AdvEnd => "ST09上阻挡下到位", Q_RetEnd => "ST09上阻挡上到位", Q_AdvLS =>, Q_RetLS =>, Q_AdvSL => "ST09上阻挡下降", Q_RetSL =>, Q_FoBraRel =>, Q_AdvTiOvErr => "Com_DB".K04.ValAdvTiOver[16], Q_RetTiOvErr => "Com_DB".K04.ValRetTiOver[16], Q_SensorsErr => "Com_DB".K04.ValSensALM[16], Q_SenCroErr => "Com_DB".K04.ValSenCroALM[16])
   END_RUNG
   RUNG wire#powerrail
      Contact( "ST09上阻挡下指令自动" )
   END_RUNG wire#w3
   RUNG wire#powerrail
      Contact( "ST09上阻挡上指令自动" )
   END_RUNG wire#w4
   RUNG wire#powerrail
      Contact( "ST09上阻挡下指令手动" )
   END_RUNG wire#w5
   RUNG wire#powerrail
      Contact( "ST09上阻挡上指令手动" )
   END_RUNG wire#w6
   RUNG wire#powerrail
      Contact( "Com_DB".K06.AdvCond_Val[16] )
   END_RUNG wire#w7
   RUNG wire#powerrail
      Contact( "Com_DB".K06.RetCond_Val[16] )
   END_RUNG wire#w8
   RUNG wire#powerrail
      Contact( "ST09上阻挡下降端" )
   END_RUNG wire#w9
   RUNG wire#powerrail
      Contact( "ST09上阻挡上升端" )
   END_RUNG wire#w10
   RUNG wire#powerrail
      Contact( "Fault_Rest" )
   END_RUNG wire#w11
   RUNG wire#powerrail
      Contact( "ManMode" )
   END_RUNG wire#w12
   // the same network as SCL:
   "Com_DB".K06.AdvCond_Val[16] := "ManMode" OR "AutoMode";
   "Com_DB".K06.RetCond_Val[16] := "ManMode" OR "AutoMode";
   #F100_Val_Instance16(I_AutoAdv := "ST09上阻挡下指令自动",   // "F100_Val"
                        I_AutoRet := "ST09上阻挡上指令自动",
                        I_ManAdv := "ST09上阻挡下指令手动",
                        I_ManRet := "ST09上阻挡上指令手动",
                        I_AdvCond := "Com_DB".K06.AdvCond_Val[16],
                        I_RetCond := "Com_DB".K06.RetCond_Val[16],
                        I_AdvLS := "ST09上阻挡下降端",
                        I_RetLS := "ST09上阻挡上升端",
                        IW_AdvTime := T#0.5S,
                        IW_RetTime := T#0.5S,
                        IW_AdvTimeOver := T#10S,
                        IW_RetTimeOver := T#10S,
                        I_Rest := "Fault_Rest",
                        I_ManMode := "ManMode",
                        IW_ConMode := 00,
                        Q_AdvEnd => "ST09上阻挡下到位",
                        Q_RetEnd => "ST09上阻挡上到位",
                        Q_AdvSL => "ST09上阻挡下降",
                        Q_AdvTiOvErr => "Com_DB".K04.ValAdvTiOver[16],
                        Q_RetTiOvErr => "Com_DB".K04.ValRetTiOver[16],
                        Q_SensorsErr => "Com_DB".K04.ValSensALM[16],
                        Q_SenCroErr => "Com_DB".K04.ValSenCroALM[16]);
END_REGION

REGION Network 17: 阀17 ST10上阻挡
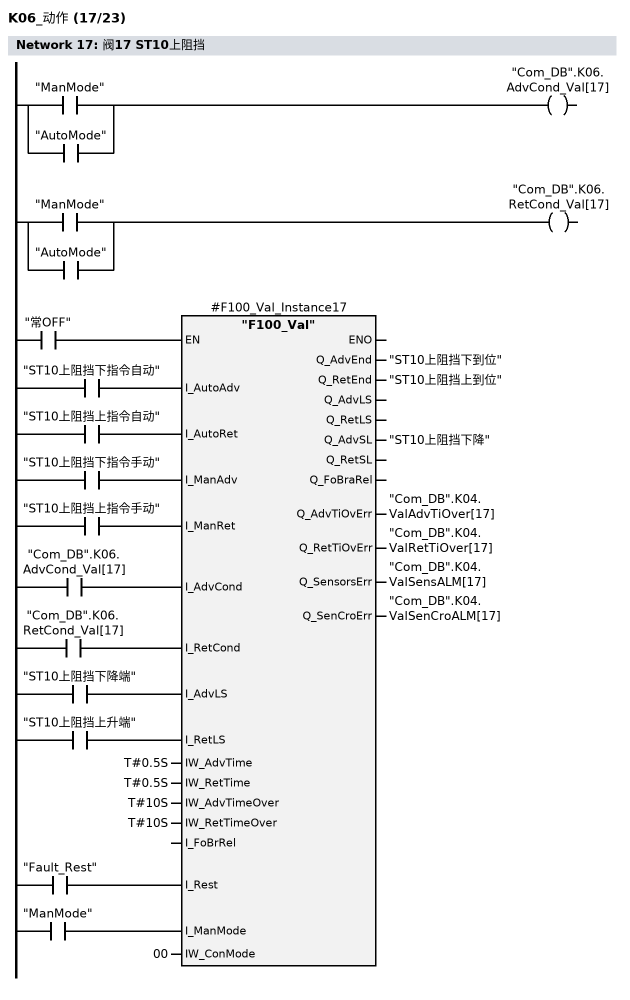
   RUNG wire#powerrail
      Contact( "ManMode" )
      wire#w1
      Coil( "Com_DB".K06.AdvCond_Val[17] )
   END_RUNG
   RUNG wire#powerrail
      Contact( "AutoMode" )
   END_RUNG wire#w1
   RUNG wire#powerrail
      Contact( "ManMode" )
      wire#w2
      Coil( "Com_DB".K06.RetCond_Val[17] )
   END_RUNG
   RUNG wire#powerrail
      Contact( "AutoMode" )
   END_RUNG wire#w2
   RUNG wire#powerrail
      Contact( "常OFF" )
      #F100_Val_Instance17(I_AutoAdv := wire#w3, I_AutoRet := wire#w4, I_ManAdv := wire#w5, I_ManRet := wire#w6, I_AdvCond := wire#w7, I_RetCond := wire#w8, I_AdvLS := wire#w9, I_RetLS := wire#w10, I_Rest := wire#w11, I_ManMode := wire#w12, IW_AdvTime := T#0.5S, IW_RetTime := T#0.5S, IW_AdvTimeOver := T#10S, IW_RetTimeOver := T#10S, I_FoBrRel :=, IW_ConMode := 00, Q_AdvEnd => "ST10上阻挡下到位", Q_RetEnd => "ST10上阻挡上到位", Q_AdvLS =>, Q_RetLS =>, Q_AdvSL => "ST10上阻挡下降", Q_RetSL =>, Q_FoBraRel =>, Q_AdvTiOvErr => "Com_DB".K04.ValAdvTiOver[17], Q_RetTiOvErr => "Com_DB".K04.ValRetTiOver[17], Q_SensorsErr => "Com_DB".K04.ValSensALM[17], Q_SenCroErr => "Com_DB".K04.ValSenCroALM[17])
   END_RUNG
   RUNG wire#powerrail
      Contact( "ST10上阻挡下指令自动" )
   END_RUNG wire#w3
   RUNG wire#powerrail
      Contact( "ST10上阻挡上指令自动" )
   END_RUNG wire#w4
   RUNG wire#powerrail
      Contact( "ST10上阻挡下指令手动" )
   END_RUNG wire#w5
   RUNG wire#powerrail
      Contact( "ST10上阻挡上指令手动" )
   END_RUNG wire#w6
   RUNG wire#powerrail
      Contact( "Com_DB".K06.AdvCond_Val[17] )
   END_RUNG wire#w7
   RUNG wire#powerrail
      Contact( "Com_DB".K06.RetCond_Val[17] )
   END_RUNG wire#w8
   RUNG wire#powerrail
      Contact( "ST10上阻挡下降端" )
   END_RUNG wire#w9
   RUNG wire#powerrail
      Contact( "ST10上阻挡上升端" )
   END_RUNG wire#w10
   RUNG wire#powerrail
      Contact( "Fault_Rest" )
   END_RUNG wire#w11
   RUNG wire#powerrail
      Contact( "ManMode" )
   END_RUNG wire#w12
   // the same network as SCL:
   "Com_DB".K06.AdvCond_Val[17] := "ManMode" OR "AutoMode";
   "Com_DB".K06.RetCond_Val[17] := "ManMode" OR "AutoMode";
   IF "常OFF" THEN
       #F100_Val_Instance17(I_AutoAdv := "ST10上阻挡下指令自动",   // "F100_Val"
                            I_AutoRet := "ST10上阻挡上指令自动",
                            I_ManAdv := "ST10上阻挡下指令手动",
                            I_ManRet := "ST10上阻挡上指令手动",
                            I_AdvCond := "Com_DB".K06.AdvCond_Val[17],
                            I_RetCond := "Com_DB".K06.RetCond_Val[17],
                            I_AdvLS := "ST10上阻挡下降端",
                            I_RetLS := "ST10上阻挡上升端",
                            IW_AdvTime := T#0.5S,
                            IW_RetTime := T#0.5S,
                            IW_AdvTimeOver := T#10S,
                            IW_RetTimeOver := T#10S,
                            I_Rest := "Fault_Rest",
                            I_ManMode := "ManMode",
                            IW_ConMode := 00,
                            Q_AdvEnd => "ST10上阻挡下到位",
                            Q_RetEnd => "ST10上阻挡上到位",
                            Q_AdvSL => "ST10上阻挡下降",
                            Q_AdvTiOvErr => "Com_DB".K04.ValAdvTiOver[17],
                            Q_RetTiOvErr => "Com_DB".K04.ValRetTiOver[17],
                            Q_SensorsErr => "Com_DB".K04.ValSensALM[17],
                            Q_SenCroErr => "Com_DB".K04.ValSenCroALM[17]);
   END_IF;
END_REGION

REGION Network 18: 阀18 ST11上阻挡
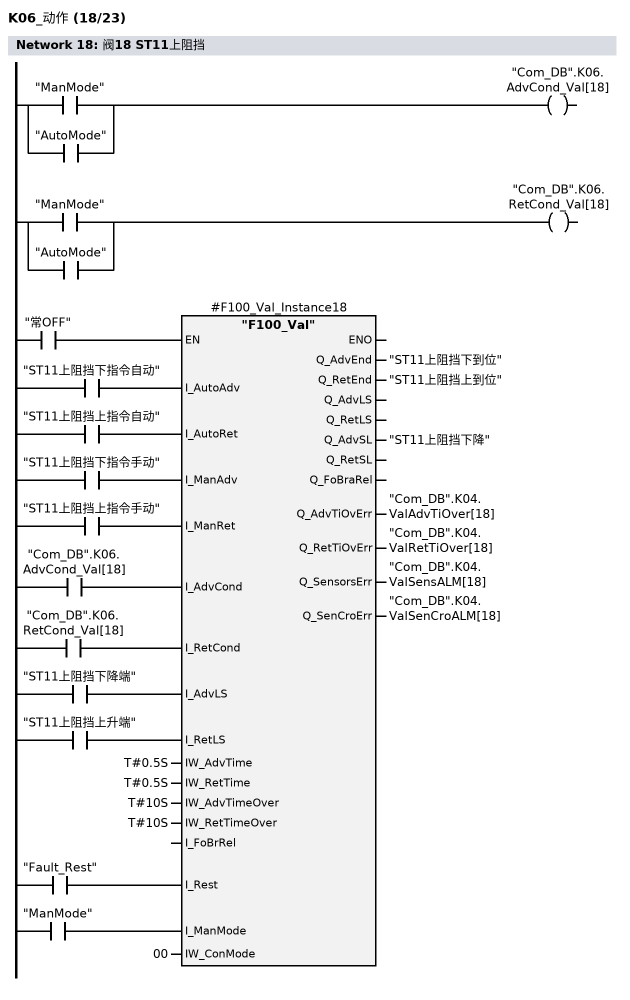
   RUNG wire#powerrail
      Contact( "ManMode" )
      wire#w1
      Coil( "Com_DB".K06.AdvCond_Val[18] )
   END_RUNG
   RUNG wire#powerrail
      Contact( "AutoMode" )
   END_RUNG wire#w1
   RUNG wire#powerrail
      Contact( "ManMode" )
      wire#w2
      Coil( "Com_DB".K06.RetCond_Val[18] )
   END_RUNG
   RUNG wire#powerrail
      Contact( "AutoMode" )
   END_RUNG wire#w2
   RUNG wire#powerrail
      Contact( "常OFF" )
      #F100_Val_Instance18(I_AutoAdv := wire#w3, I_AutoRet := wire#w4, I_ManAdv := wire#w5, I_ManRet := wire#w6, I_AdvCond := wire#w7, I_RetCond := wire#w8, I_AdvLS := wire#w9, I_RetLS := wire#w10, I_Rest := wire#w11, I_ManMode := wire#w12, IW_AdvTime := T#0.5S, IW_RetTime := T#0.5S, IW_AdvTimeOver := T#10S, IW_RetTimeOver := T#10S, I_FoBrRel :=, IW_ConMode := 00, Q_AdvEnd => "ST11上阻挡下到位", Q_RetEnd => "ST11上阻挡上到位", Q_AdvLS =>, Q_RetLS =>, Q_AdvSL => "ST11上阻挡下降", Q_RetSL =>, Q_FoBraRel =>, Q_AdvTiOvErr => "Com_DB".K04.ValAdvTiOver[18], Q_RetTiOvErr => "Com_DB".K04.ValRetTiOver[18], Q_SensorsErr => "Com_DB".K04.ValSensALM[18], Q_SenCroErr => "Com_DB".K04.ValSenCroALM[18])
   END_RUNG
   RUNG wire#powerrail
      Contact( "ST11上阻挡下指令自动" )
   END_RUNG wire#w3
   RUNG wire#powerrail
      Contact( "ST11上阻挡上指令自动" )
   END_RUNG wire#w4
   RUNG wire#powerrail
      Contact( "ST11上阻挡下指令手动" )
   END_RUNG wire#w5
   RUNG wire#powerrail
      Contact( "ST11上阻挡上指令手动" )
   END_RUNG wire#w6
   RUNG wire#powerrail
      Contact( "Com_DB".K06.AdvCond_Val[18] )
   END_RUNG wire#w7
   RUNG wire#powerrail
      Contact( "Com_DB".K06.RetCond_Val[18] )
   END_RUNG wire#w8
   RUNG wire#powerrail
      Contact( "ST11上阻挡下降端" )
   END_RUNG wire#w9
   RUNG wire#powerrail
      Contact( "ST11上阻挡上升端" )
   END_RUNG wire#w10
   RUNG wire#powerrail
      Contact( "Fault_Rest" )
   END_RUNG wire#w11
   RUNG wire#powerrail
      Contact( "ManMode" )
   END_RUNG wire#w12
   // the same network as SCL:
   "Com_DB".K06.AdvCond_Val[18] := "ManMode" OR "AutoMode";
   "Com_DB".K06.RetCond_Val[18] := "ManMode" OR "AutoMode";
   IF "常OFF" THEN
       #F100_Val_Instance18(I_AutoAdv := "ST11上阻挡下指令自动",   // "F100_Val"
                            I_AutoRet := "ST11上阻挡上指令自动",
                            I_ManAdv := "ST11上阻挡下指令手动",
                            I_ManRet := "ST11上阻挡上指令手动",
                            I_AdvCond := "Com_DB".K06.AdvCond_Val[18],
                            I_RetCond := "Com_DB".K06.RetCond_Val[18],
                            I_AdvLS := "ST11上阻挡下降端",
                            I_RetLS := "ST11上阻挡上升端",
                            IW_AdvTime := T#0.5S,
                            IW_RetTime := T#0.5S,
                            IW_AdvTimeOver := T#10S,
                            IW_RetTimeOver := T#10S,
                            I_Rest := "Fault_Rest",
                            I_ManMode := "ManMode",
                            IW_ConMode := 00,
                            Q_AdvEnd => "ST11上阻挡下到位",
                            Q_RetEnd => "ST11上阻挡上到位",
                            Q_AdvSL => "ST11上阻挡下降",
                            Q_AdvTiOvErr => "Com_DB".K04.ValAdvTiOver[18],
                            Q_RetTiOvErr => "Com_DB".K04.ValRetTiOver[18],
                            Q_SensorsErr => "Com_DB".K04.ValSensALM[18],
                            Q_SenCroErr => "Com_DB".K04.ValSenCroALM[18]);
   END_IF;
END_REGION

REGION Network 19: 阀19 ST12上阻挡
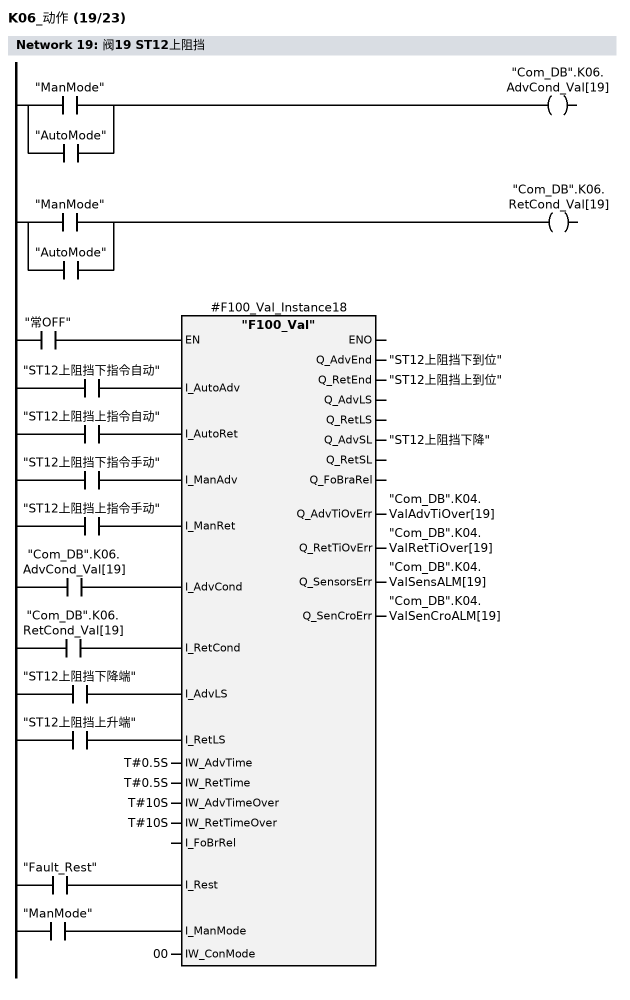
   RUNG wire#powerrail
      Contact( "ManMode" )
      wire#w1
      Coil( "Com_DB".K06.AdvCond_Val[19] )
   END_RUNG
   RUNG wire#powerrail
      Contact( "AutoMode" )
   END_RUNG wire#w1
   RUNG wire#powerrail
      Contact( "ManMode" )
      wire#w2
      Coil( "Com_DB".K06.RetCond_Val[19] )
   END_RUNG
   RUNG wire#powerrail
      Contact( "AutoMode" )
   END_RUNG wire#w2
   RUNG wire#powerrail
      Contact( "常OFF" )
      #F100_Val_Instance18(I_AutoAdv := wire#w3, I_AutoRet := wire#w4, I_ManAdv := wire#w5, I_ManRet := wire#w6, I_AdvCond := wire#w7, I_RetCond := wire#w8, I_AdvLS := wire#w9, I_RetLS := wire#w10, I_Rest := wire#w11, I_ManMode := wire#w12, IW_AdvTime := T#0.5S, IW_RetTime := T#0.5S, IW_AdvTimeOver := T#10S, IW_RetTimeOver := T#10S, I_FoBrRel :=, IW_ConMode := 00, Q_AdvEnd => "ST12上阻挡下到位", Q_RetEnd => "ST12上阻挡上到位", Q_AdvLS =>, Q_RetLS =>, Q_AdvSL => "ST12上阻挡下降", Q_RetSL =>, Q_FoBraRel =>, Q_AdvTiOvErr => "Com_DB".K04.ValAdvTiOver[19], Q_RetTiOvErr => "Com_DB".K04.ValRetTiOver[19], Q_SensorsErr => "Com_DB".K04.ValSensALM[19], Q_SenCroErr => "Com_DB".K04.ValSenCroALM[19])
   END_RUNG
   RUNG wire#powerrail
      Contact( "ST12上阻挡下指令自动" )
   END_RUNG wire#w3
   RUNG wire#powerrail
      Contact( "ST12上阻挡上指令自动" )
   END_RUNG wire#w4
   RUNG wire#powerrail
      Contact( "ST12上阻挡下指令手动" )
   END_RUNG wire#w5
   RUNG wire#powerrail
      Contact( "ST12上阻挡上指令手动" )
   END_RUNG wire#w6
   RUNG wire#powerrail
      Contact( "Com_DB".K06.AdvCond_Val[19] )
   END_RUNG wire#w7
   RUNG wire#powerrail
      Contact( "Com_DB".K06.RetCond_Val[19] )
   END_RUNG wire#w8
   RUNG wire#powerrail
      Contact( "ST12上阻挡下降端" )
   END_RUNG wire#w9
   RUNG wire#powerrail
      Contact( "ST12上阻挡上升端" )
   END_RUNG wire#w10
   RUNG wire#powerrail
      Contact( "Fault_Rest" )
   END_RUNG wire#w11
   RUNG wire#powerrail
      Contact( "ManMode" )
   END_RUNG wire#w12
   // the same network as SCL:
   "Com_DB".K06.AdvCond_Val[19] := "ManMode" OR "AutoMode";
   "Com_DB".K06.RetCond_Val[19] := "ManMode" OR "AutoMode";
   IF "常OFF" THEN
       #F100_Val_Instance18(I_AutoAdv := "ST12上阻挡下指令自动",   // "F100_Val"
                            I_AutoRet := "ST12上阻挡上指令自动",
                            I_ManAdv := "ST12上阻挡下指令手动",
                            I_ManRet := "ST12上阻挡上指令手动",
                            I_AdvCond := "Com_DB".K06.AdvCond_Val[19],
                            I_RetCond := "Com_DB".K06.RetCond_Val[19],
                            I_AdvLS := "ST12上阻挡下降端",
                            I_RetLS := "ST12上阻挡上升端",
                            IW_AdvTime := T#0.5S,
                            IW_RetTime := T#0.5S,
                            IW_AdvTimeOver := T#10S,
                            IW_RetTimeOver := T#10S,
                            I_Rest := "Fault_Rest",
                            I_ManMode := "ManMode",
                            IW_ConMode := 00,
                            Q_AdvEnd => "ST12上阻挡下到位",
                            Q_RetEnd => "ST12上阻挡上到位",
                            Q_AdvSL => "ST12上阻挡下降",
                            Q_AdvTiOvErr => "Com_DB".K04.ValAdvTiOver[19],
                            Q_RetTiOvErr => "Com_DB".K04.ValRetTiOver[19],
                            Q_SensorsErr => "Com_DB".K04.ValSensALM[19],
                            Q_SenCroErr => "Com_DB".K04.ValSenCroALM[19]);
   END_IF;
END_REGION

REGION Network 20: 变频器1-入口搬送电机
   // 滚筒控制也可以使用变频器FB库，正转上层送托盘，反转下层接托盘
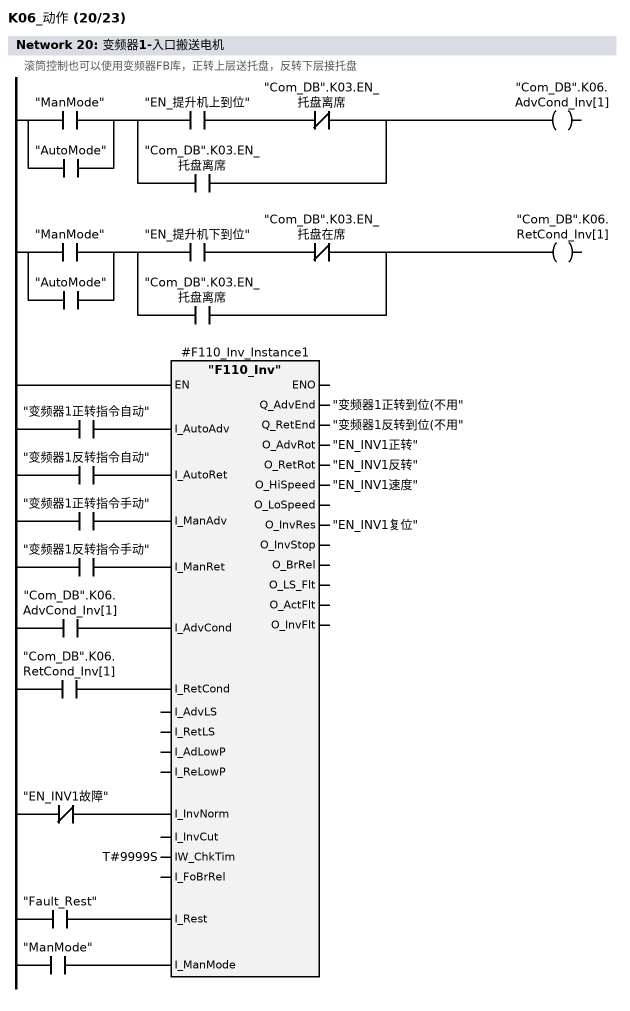
   RUNG wire#powerrail
      Contact( "ManMode" )
      wire#w1
      Contact( "EN_提升机上到位" )
      I_Contact( "Com_DB".K03.EN_托盘离席 )
      wire#w2
      Coil( "Com_DB".K06.AdvCond_Inv[1] )
   END_RUNG
   RUNG wire#powerrail
      Contact( "AutoMode" )
   END_RUNG wire#w1
   RUNG wire#w1
      Contact( "Com_DB".K03.EN_托盘离席 )
   END_RUNG wire#w2
   RUNG wire#powerrail
      Contact( "ManMode" )
      wire#w3
      Contact( "EN_提升机下到位" )
      I_Contact( "Com_DB".K03.EN_托盘在席 )
      wire#w4
      Coil( "Com_DB".K06.RetCond_Inv[1] )
   END_RUNG
   RUNG wire#powerrail
      Contact( "AutoMode" )
   END_RUNG wire#w3
   RUNG wire#w3
      Contact( "Com_DB".K03.EN_托盘离席 )
   END_RUNG wire#w4
   RUNG wire#powerrail
      #F110_Inv_Instance1(I_AutoAdv := wire#w5, I_AutoRet := wire#w6, I_ManAdv := wire#w7, I_ManRet := wire#w8, I_AdvCond := wire#w9, I_RetCond := wire#w10, I_InvNorm := wire#w11, I_Rest := wire#w12, I_ManMode := wire#w13, I_AdvLS :=, I_RetLS :=, I_AdLowP :=, I_ReLowP :=, I_InvCut :=, IW_ChkTim := T#9999S, I_FoBrRel :=, Q_AdvEnd => "变频器1正转到位(不用", Q_RetEnd => "变频器1反转到位(不用", O_AdvRot => "EN_INV1正转", O_RetRot => "EN_INV1反转", O_HiSpeed => "EN_INV1速度", O_LoSpeed =>, O_InvRes => "EN_INV1复位", O_InvStop =>, O_BrRel =>, O_LS_Flt =>, O_ActFlt =>, O_InvFlt =>)
   END_RUNG
   RUNG wire#powerrail
      Contact( "变频器1正转指令自动" )
   END_RUNG wire#w5
   RUNG wire#powerrail
      Contact( "变频器1反转指令自动" )
   END_RUNG wire#w6
   RUNG wire#powerrail
      Contact( "变频器1正转指令手动" )
   END_RUNG wire#w7
   RUNG wire#powerrail
      Contact( "变频器1反转指令手动" )
   END_RUNG wire#w8
   RUNG wire#powerrail
      Contact( "Com_DB".K06.AdvCond_Inv[1] )
   END_RUNG wire#w9
   RUNG wire#powerrail
      Contact( "Com_DB".K06.RetCond_Inv[1] )
   END_RUNG wire#w10
   RUNG wire#powerrail
      I_Contact( "EN_INV1故障" )
   END_RUNG wire#w11
   RUNG wire#powerrail
      Contact( "Fault_Rest" )
   END_RUNG wire#w12
   RUNG wire#powerrail
      Contact( "ManMode" )
   END_RUNG wire#w13
   // the same network as SCL:
   "Com_DB".K06.AdvCond_Inv[1] := ("ManMode" OR "AutoMode") AND (("EN_提升机上到位" AND NOT "Com_DB".K03.EN_托盘离席) OR "Com_DB".K03.EN_托盘离席);
   "Com_DB".K06.RetCond_Inv[1] := ("ManMode" OR "AutoMode") AND (("EN_提升机下到位" AND NOT "Com_DB".K03.EN_托盘在席) OR "Com_DB".K03.EN_托盘离席);
   #F110_Inv_Instance1(I_AutoAdv := "变频器1正转指令自动",   // "F110_Inv"
                       I_AutoRet := "变频器1反转指令自动",
                       I_ManAdv := "变频器1正转指令手动",
                       I_ManRet := "变频器1反转指令手动",
                       I_AdvCond := "Com_DB".K06.AdvCond_Inv[1],
                       I_RetCond := "Com_DB".K06.RetCond_Inv[1],
                       I_InvNorm := NOT "EN_INV1故障",
                       IW_ChkTim := T#9999S,
                       I_Rest := "Fault_Rest",
                       I_ManMode := "ManMode",
                       Q_AdvEnd => "变频器1正转到位(不用",
                       Q_RetEnd => "变频器1反转到位(不用",
                       O_AdvRot => "EN_INV1正转",
                       O_RetRot => "EN_INV1反转",
                       O_HiSpeed => "EN_INV1速度",
                       O_InvRes => "EN_INV1复位");
END_REGION

REGION Network 21: 变频器2 出口搬送电机
   // 正转上层J接托盘，反转下层送托盘
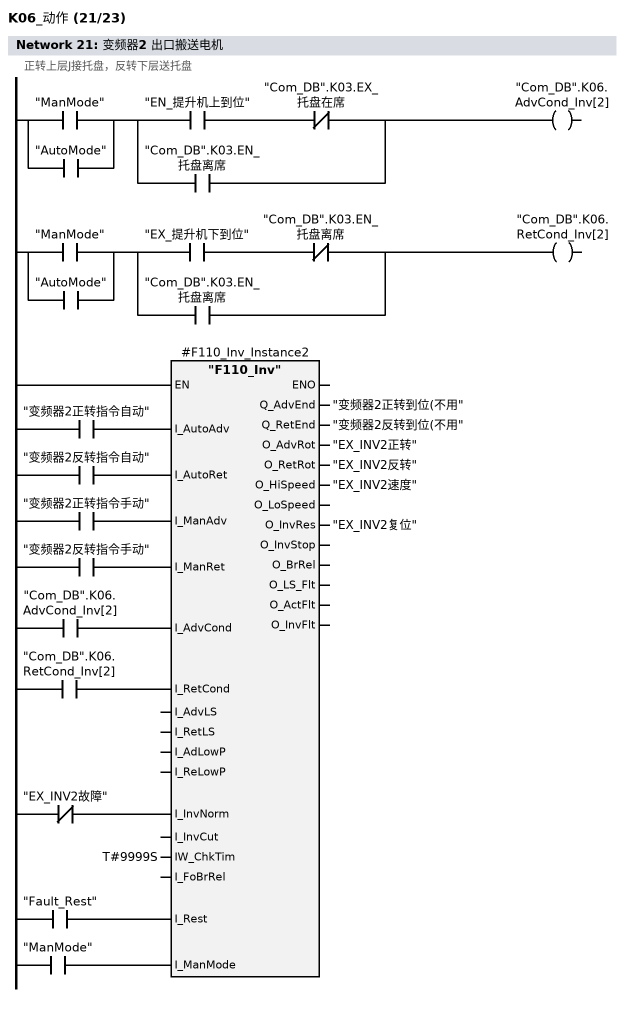
   RUNG wire#powerrail
      Contact( "ManMode" )
      wire#w1
      Contact( "EN_提升机上到位" )
      I_Contact( "Com_DB".K03.EX_托盘在席 )
      wire#w2
      Coil( "Com_DB".K06.AdvCond_Inv[2] )
   END_RUNG
   RUNG wire#powerrail
      Contact( "AutoMode" )
   END_RUNG wire#w1
   RUNG wire#w1
      Contact( "Com_DB".K03.EN_托盘离席 )
   END_RUNG wire#w2
   RUNG wire#powerrail
      Contact( "ManMode" )
      wire#w3
      Contact( "EX_提升机下到位" )
      I_Contact( "Com_DB".K03.EN_托盘离席 )
      wire#w4
      Coil( "Com_DB".K06.RetCond_Inv[2] )
   END_RUNG
   RUNG wire#powerrail
      Contact( "AutoMode" )
   END_RUNG wire#w3
   RUNG wire#w3
      Contact( "Com_DB".K03.EN_托盘离席 )
   END_RUNG wire#w4
   RUNG wire#powerrail
      #F110_Inv_Instance2(I_AutoAdv := wire#w5, I_AutoRet := wire#w6, I_ManAdv := wire#w7, I_ManRet := wire#w8, I_AdvCond := wire#w9, I_RetCond := wire#w10, I_InvNorm := wire#w11, I_Rest := wire#w12, I_ManMode := wire#w13, I_AdvLS :=, I_RetLS :=, I_AdLowP :=, I_ReLowP :=, I_InvCut :=, IW_ChkTim := T#9999S, I_FoBrRel :=, Q_AdvEnd => "变频器2正转到位(不用", Q_RetEnd => "变频器2反转到位(不用", O_AdvRot => "EX_INV2正转", O_RetRot => "EX_INV2反转", O_HiSpeed => "EX_INV2速度", O_LoSpeed =>, O_InvRes => "EX_INV2复位", O_InvStop =>, O_BrRel =>, O_LS_Flt =>, O_ActFlt =>, O_InvFlt =>)
   END_RUNG
   RUNG wire#powerrail
      Contact( "变频器2正转指令自动" )
   END_RUNG wire#w5
   RUNG wire#powerrail
      Contact( "变频器2反转指令自动" )
   END_RUNG wire#w6
   RUNG wire#powerrail
      Contact( "变频器2正转指令手动" )
   END_RUNG wire#w7
   RUNG wire#powerrail
      Contact( "变频器2反转指令手动" )
   END_RUNG wire#w8
   RUNG wire#powerrail
      Contact( "Com_DB".K06.AdvCond_Inv[2] )
   END_RUNG wire#w9
   RUNG wire#powerrail
      Contact( "Com_DB".K06.RetCond_Inv[2] )
   END_RUNG wire#w10
   RUNG wire#powerrail
      I_Contact( "EX_INV2故障" )
   END_RUNG wire#w11
   RUNG wire#powerrail
      Contact( "Fault_Rest" )
   END_RUNG wire#w12
   RUNG wire#powerrail
      Contact( "ManMode" )
   END_RUNG wire#w13
   // the same network as SCL:
   "Com_DB".K06.AdvCond_Inv[2] := ("ManMode" OR "AutoMode") AND (("EN_提升机上到位" AND NOT "Com_DB".K03.EX_托盘在席) OR "Com_DB".K03.EN_托盘离席);
   "Com_DB".K06.RetCond_Inv[2] := ("ManMode" OR "AutoMode") AND (("EX_提升机下到位" AND NOT "Com_DB".K03.EN_托盘离席) OR "Com_DB".K03.EN_托盘离席);
   #F110_Inv_Instance2(I_AutoAdv := "变频器2正转指令自动",   // "F110_Inv"
                       I_AutoRet := "变频器2反转指令自动",
                       I_ManAdv := "变频器2正转指令手动",
                       I_ManRet := "变频器2反转指令手动",
                       I_AdvCond := "Com_DB".K06.AdvCond_Inv[2],
                       I_RetCond := "Com_DB".K06.RetCond_Inv[2],
                       I_InvNorm := NOT "EX_INV2故障",
                       IW_ChkTim := T#9999S,
                       I_Rest := "Fault_Rest",
                       I_ManMode := "ManMode",
                       Q_AdvEnd => "变频器2正转到位(不用",
                       Q_RetEnd => "变频器2反转到位(不用",
                       O_AdvRot => "EX_INV2正转",
                       O_RetRot => "EX_INV2反转",
                       O_HiSpeed => "EX_INV2速度",
                       O_InvRes => "EX_INV2复位");
END_REGION

REGION Network 22: 变频器3/5 前段/后段上层搬送电机，因为上层变频器条件一致，功能一致。共用1个FB
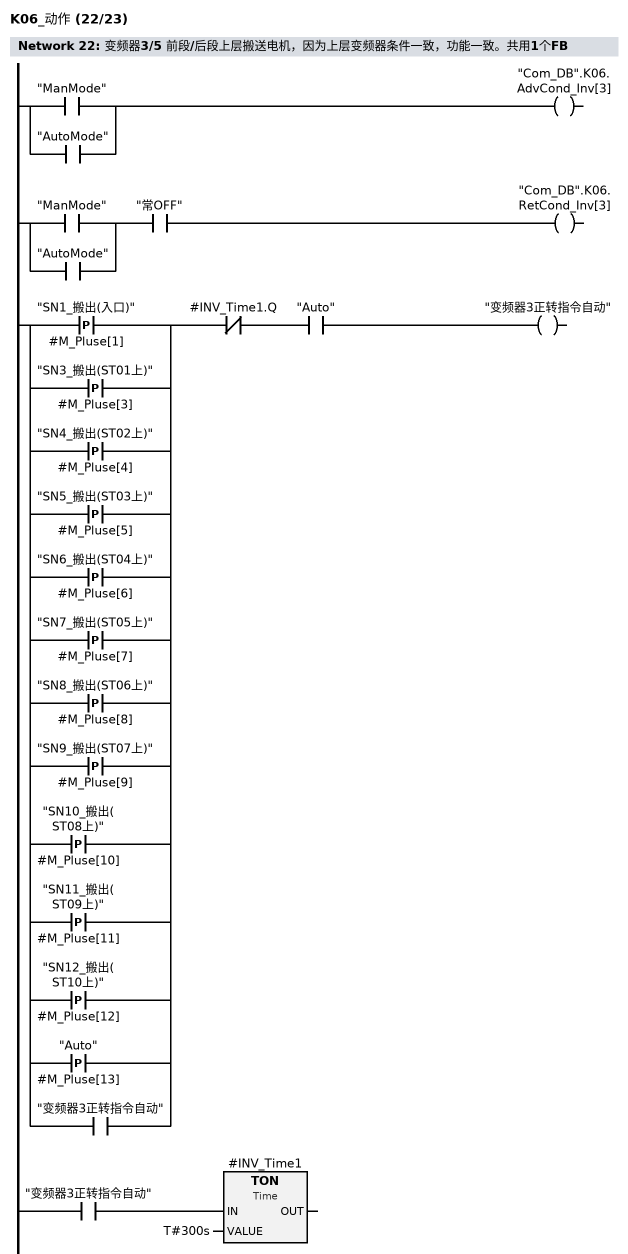
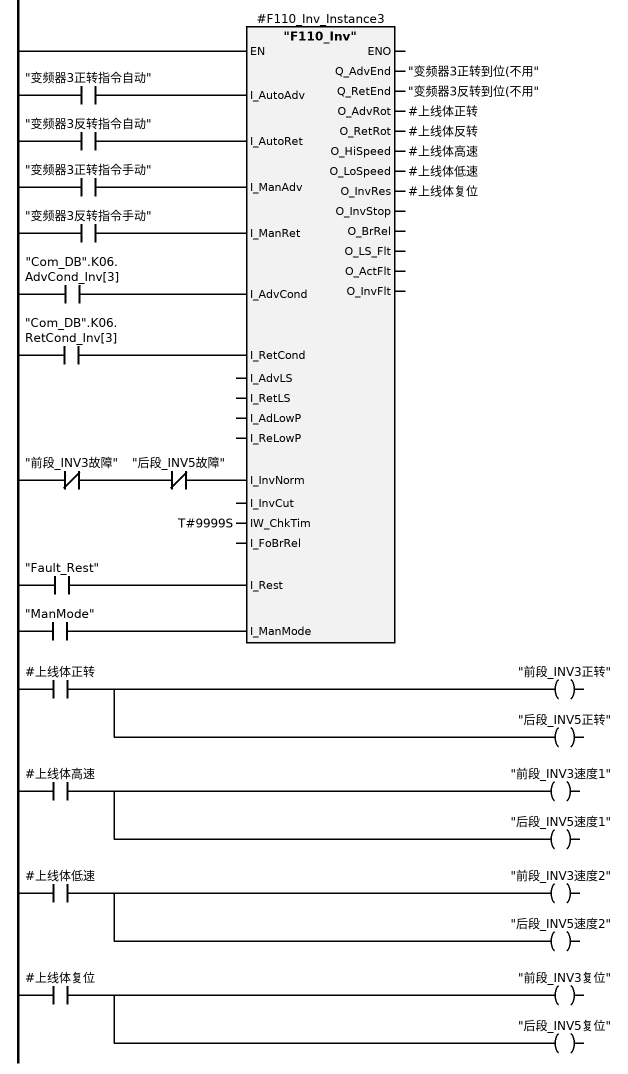
   "Com_DB".K06.AdvCond_Inv[3] := "ManMode" OR "AutoMode";
   "Com_DB".K06.RetCond_Inv[3] := ("ManMode" OR "AutoMode") AND "常OFF";
   #_w1 := "SN1_搬出(入口)" AND NOT #M_Pluse[1];   // rising edge of "SN1_搬出(入口)"
   #M_Pluse[1] := "SN1_搬出(入口)";
   #_w2 := "SN3_搬出(ST01上)" AND NOT #M_Pluse[3];   // rising edge of "SN3_搬出(ST01上)"
   #M_Pluse[3] := "SN3_搬出(ST01上)";
   #_w3 := "SN4_搬出(ST02上)" AND NOT #M_Pluse[4];   // rising edge of "SN4_搬出(ST02上)"
   #M_Pluse[4] := "SN4_搬出(ST02上)";
   #_w4 := "SN5_搬出(ST03上)" AND NOT #M_Pluse[5];   // rising edge of "SN5_搬出(ST03上)"
   #M_Pluse[5] := "SN5_搬出(ST03上)";
   #_w5 := "SN6_搬出(ST04上)" AND NOT #M_Pluse[6];   // rising edge of "SN6_搬出(ST04上)"
   #M_Pluse[6] := "SN6_搬出(ST04上)";
   #_w6 := "SN7_搬出(ST05上)" AND NOT #M_Pluse[7];   // rising edge of "SN7_搬出(ST05上)"
   #M_Pluse[7] := "SN7_搬出(ST05上)";
   #_w7 := "SN8_搬出(ST06上)" AND NOT #M_Pluse[8];   // rising edge of "SN8_搬出(ST06上)"
   #M_Pluse[8] := "SN8_搬出(ST06上)";
   #_w8 := "SN9_搬出(ST07上)" AND NOT #M_Pluse[9];   // rising edge of "SN9_搬出(ST07上)"
   #M_Pluse[9] := "SN9_搬出(ST07上)";
   #_w9 := "SN10_搬出(ST08上)" AND NOT #M_Pluse[10];   // rising edge of "SN10_搬出(ST08上)"
   #M_Pluse[10] := "SN10_搬出(ST08上)";
   #_w10 := "SN11_搬出(ST09上)" AND NOT #M_Pluse[11];   // rising edge of "SN11_搬出(ST09上)"
   #M_Pluse[11] := "SN11_搬出(ST09上)";
   #_w11 := "SN12_搬出(ST10上)" AND NOT #M_Pluse[12];   // rising edge of "SN12_搬出(ST10上)"
   #M_Pluse[12] := "SN12_搬出(ST10上)";
   #_w12 := "Auto" AND NOT #M_Pluse[13];   // rising edge of "Auto"
   #M_Pluse[13] := "Auto";
   "变频器3正转指令自动" := (#_w1 OR #_w2 OR #_w3 OR #_w4 OR #_w5 OR #_w6 OR #_w7 OR #_w8 OR #_w9 OR #_w10 OR #_w11 OR #_w12 OR "变频器3正转指令自动") AND NOT #INV_Time1.Q AND "Auto";
   #INV_Time1.TON(IN := "变频器3正转指令自动", PT := T#300s);   // TON coil
   #F110_Inv_Instance3(I_AutoAdv := "变频器3正转指令自动",   // "F110_Inv"
                       I_AutoRet := "变频器3反转指令自动",
                       I_ManAdv := "变频器3正转指令手动",
                       I_ManRet := "变频器3反转指令手动",
                       I_AdvCond := "Com_DB".K06.AdvCond_Inv[3],
                       I_RetCond := "Com_DB".K06.RetCond_Inv[3],
                       I_InvNorm := NOT "前段_INV3故障" AND NOT "后段_INV5故障",
                       IW_ChkTim := T#9999S,
                       I_Rest := "Fault_Rest",
                       I_ManMode := "ManMode",
                       Q_AdvEnd => "变频器3正转到位(不用",
                       Q_RetEnd => "变频器3反转到位(不用",
                       O_AdvRot => #上线体正转,
                       O_RetRot => #上线体反转,
                       O_HiSpeed => #上线体高速,
                       O_LoSpeed => #上线体低速,
                       O_InvRes => #上线体复位);
   "前段_INV3正转" := #上线体正转;
   "后段_INV5正转" := #上线体正转;
   "前段_INV3速度1" := #上线体高速;
   "后段_INV5速度1" := #上线体高速;
   "前段_INV3速度2" := #上线体低速;
   "后段_INV5速度2" := #上线体低速;
   "前段_INV3复位" := #上线体复位;
   "后段_INV5复位" := #上线体复位;
END_REGION

REGION Network 23: 变频器4/6前段/后段下层搬送电机。因为上层变频器条件一致，功能一致。共用1个FB
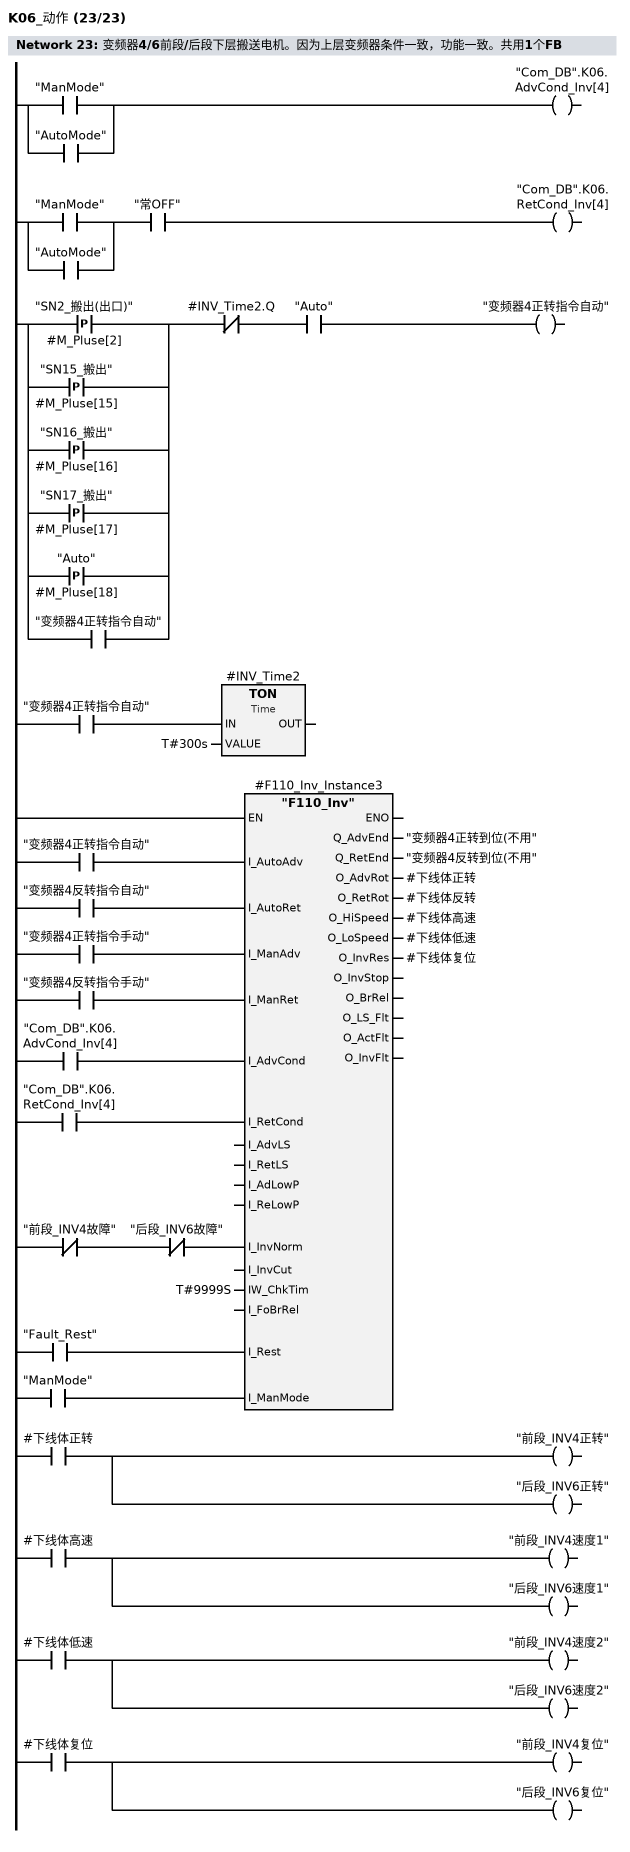
   "Com_DB".K06.AdvCond_Inv[4] := "ManMode" OR "AutoMode";
   "Com_DB".K06.RetCond_Inv[4] := ("ManMode" OR "AutoMode") AND "常OFF";
   #_w1 := "SN2_搬出(出口)" AND NOT #M_Pluse[2];   // rising edge of "SN2_搬出(出口)"
   #M_Pluse[2] := "SN2_搬出(出口)";
   #_w2 := "SN15_搬出" AND NOT #M_Pluse[15];   // rising edge of "SN15_搬出"
   #M_Pluse[15] := "SN15_搬出";
   #_w3 := "SN16_搬出" AND NOT #M_Pluse[16];   // rising edge of "SN16_搬出"
   #M_Pluse[16] := "SN16_搬出";
   #_w4 := "SN17_搬出" AND NOT #M_Pluse[17];   // rising edge of "SN17_搬出"
   #M_Pluse[17] := "SN17_搬出";
   #_w5 := "Auto" AND NOT #M_Pluse[18];   // rising edge of "Auto"
   #M_Pluse[18] := "Auto";
   "变频器4正转指令自动" := (#_w1 OR #_w2 OR #_w3 OR #_w4 OR #_w5 OR "变频器4正转指令自动") AND NOT #INV_Time2.Q AND "Auto";
   #INV_Time2.TON(IN := "变频器4正转指令自动", PT := T#300s);   // TON coil
   #F110_Inv_Instance3(I_AutoAdv := "变频器4正转指令自动",   // "F110_Inv"
                       I_AutoRet := "变频器4反转指令自动",
                       I_ManAdv := "变频器4正转指令手动",
                       I_ManRet := "变频器4反转指令手动",
                       I_AdvCond := "Com_DB".K06.AdvCond_Inv[4],
                       I_RetCond := "Com_DB".K06.RetCond_Inv[4],
                       I_InvNorm := NOT "前段_INV4故障" AND NOT "后段_INV6故障",
                       IW_ChkTim := T#9999S,
                       I_Rest := "Fault_Rest",
                       I_ManMode := "ManMode",
                       Q_AdvEnd => "变频器4正转到位(不用",
                       Q_RetEnd => "变频器4反转到位(不用",
                       O_AdvRot => #下线体正转,
                       O_RetRot => #下线体反转,
                       O_HiSpeed => #下线体高速,
                       O_LoSpeed => #下线体低速,
                       O_InvRes => #下线体复位);
   "前段_INV4正转" := #下线体正转;
   "后段_INV6正转" := #下线体正转;
   "前段_INV4速度1" := #下线体高速;
   "后段_INV6速度1" := #下线体高速;
   "前段_INV4速度2" := #下线体低速;
   "后段_INV6速度2" := #下线体低速;
   "前段_INV4复位" := #下线体复位;
   "后段_INV6复位" := #下线体复位;
END_REGION
END_FUNCTION_BLOCK
